   1:  PR[91,3] = PR[90,3] + 50.738;
   1:L PR[91] R[100]mm/sec CNT100;
   1:  PR[91,1] = PR[90,1] + 22.641;
   1:  PR[91,2] = PR[90,2] + -11.815;
   1:  PR[91,3] = PR[90,3] + 50.748;
   1:L PR[91] R[100]mm/sec CNT100;
   1:  PR[91,1] = PR[90,1] + 23.256;
   1:  PR[91,2] = PR[90,2] + -10.902;
   1:  PR[91,3] = PR[90,3] + 50.757;
   1:L PR[91] R[100]mm/sec CNT100;
   1:  PR[91,1] = PR[90,1] + 23.822;
   1:  PR[91,2] = PR[90,2] + -9.962;
   1:  PR[91,3] = PR[90,3] + 50.767;
   1:L PR[91] R[100]mm/sec CNT100;
   1:  PR[91,1] = PR[90,1] + 24.339;
   1:  PR[91,2] = PR[90,2] + -8.997;
   1:  PR[91,3] = PR[90,3] + 50.776;
   1:L PR[91] R[100]mm/sec CNT100;
   1:  PR[91,1] = PR[90,1] + 24.805;
   1:  PR[91,2] = PR[90,2] + -8.010;
   1:  PR[91,3] = PR[90,3] + 50.785;
   1:L PR[91] R[100]mm/sec CNT100;
   1:  PR[91,1] = PR[90,1] + 25.218;
   1:  PR[91,2] = PR[90,2] + -7.005;
   1:  PR[91,3] = PR[90,3] + 50.795;
   1:L PR[91] R[100]mm/sec CNT100;
   1:  PR[91,1] = PR[90,1] + 25.578;
   1:  PR[91,2] = PR[90,2] + -5.984;
   1:  PR[91,3] = PR[90,3] + 50.804;
   1:L PR[91] R[100]mm/sec CNT100;
   1:  PR[91,1] = PR[90,1] + 25.884;
   1:  PR[91,2] = PR[90,2] + -4.948;
   1:  PR[91,3] = PR[90,3] + 50.813;
   1:L PR[91] R[100]mm/sec CNT100;
   1:  PR[91,1] = PR[90,1] + 26.135;
   1:  PR[91,2] = PR[90,2] + -3.900;
   1:  PR[91,3] = PR[90,3] + 50.822;
   1:L PR[91] R[100]mm/sec CNT100;
   1:  PR[91,1] = PR[90,1] + 26.331;
   1:  PR[91,2] = PR[90,2] + -2.838;
   1:  PR[91,3] = PR[90,3] + 50.832;
   1:L PR[91] R[100]mm/sec CNT100;
   1:  PR[91,1] = PR[90,1] + 26.472;
   1:  PR[91,2] = PR[90,2] + -1.762;
   1:  PR[91,3] = PR[90,3] + 50.841;
   1:L PR[91] R[100]mm/sec CNT100;
   1:  PR[91,1] = PR[90,1] + 26.556;
   1:  PR[91,2] = PR[90,2] + -0.674;
   1:  PR[91,3] = PR[90,3] + 50.850;
   1:L PR[91] R[100]mm/sec CNT100;
   1:  PR[91,1] = PR[90,1] + 26.584;
   1:  PR[91,2] = PR[90,2] + 0.428;
   1:  PR[91,3] = PR[90,3] + 50.860;
   1:L PR[91] R[100]mm/sec CNT100;
   1:  PR[91,1] = PR[90,1] + 26.556;
   1:  PR[91,2] = PR[90,2] + 1.529;
   1:  PR[91,3] = PR[90,3] + 50.869;
   1:L PR[91] R[100]mm/sec CNT100;
   1:  PR[91,1] = PR[90,1] + 26.472;
   1:  PR[91,2] = PR[90,2] + 2.617;
   1:  PR[91,3] = PR[90,3] + 50.878;
   1:L PR[91] R[100]mm/sec CNT100;
   1:  PR[91,1] = PR[90,1] + 26.331;
   1:  PR[91,2] = PR[90,2] + 3.692;
   1:  PR[91,3] = PR[90,3] + 50.888;
   1:L PR[91] R[100]mm/sec CNT100;
   1:  PR[91,1] = PR[90,1] + 26.135;
   1:  PR[91,2] = PR[90,2] + 4.755;
   1:  PR[91,3] = PR[90,3] + 50.897;
   1:L PR[91] R[100]mm/sec CNT100;
   1:  PR[91,1] = PR[90,1] + 25.884;
   1:  PR[91,2] = PR[90,2] + 5.803;
   1:  PR[91,3] = PR[90,3] + 50.906;
   1:L PR[91] R[100]mm/sec CNT100;
   1:  PR[91,1] = PR[90,1] + 25.578;
   1:  PR[91,2] = PR[90,2] + 6.839;
   1:  PR[91,3] = PR[90,3] + 50.915;
   1:L PR[91] R[100]mm/sec CNT100;
   1:  PR[91,1] = PR[90,1] + 25.218;
   1:  PR[91,2] = PR[90,2] + 7.860;
   1:  PR[91,3] = PR[90,3] + 50.925;
   1:L PR[91] R[100]mm/sec CNT100;
   1:  PR[91,1] = PR[90,1] + 24.805;
   1:  PR[91,2] = PR[90,2] + 8.864;
   1:  PR[91,3] = PR[90,3] + 50.934;
   1:L PR[91] R[100]mm/sec CNT100;
   1:  PR[91,1] = PR[90,1] + 24.339;
   1:  PR[91,2] = PR[90,2] + 9.851;
   1:  PR[91,3] = PR[90,3] + 50.943;
   1:L PR[91] R[100]mm/sec CNT100;
   1:  PR[91,1] = PR[90,1] + 23.823;
   1:  PR[91,2] = PR[90,2] + 10.817;
   1:  PR[91,3] = PR[90,3] + 50.953;
   1:L PR[91] R[100]mm/sec CNT100;
   1:  PR[91,1] = PR[90,1] + 23.256;
   1:  PR[91,2] = PR[90,2] + 11.757;
   1:  PR[91,3] = PR[90,3] + 50.962;
   1:L PR[91] R[100]mm/sec CNT100;
   1:  PR[91,1] = PR[90,1] + 22.642;
   1:  PR[91,2] = PR[90,2] + 12.669;
   1:  PR[91,3] = PR[90,3] + 50.971;
   1:L PR[91] R[100]mm/sec CNT100;
   1:  PR[91,1] = PR[90,1] + 21.980;
   1:  PR[91,2] = PR[90,2] + 13.551;
   1:  PR[91,3] = PR[90,3] + 50.981;
   1:L PR[91] R[100]mm/sec CNT100;
   1:  PR[91,1] = PR[90,1] + 21.273;
   1:  PR[91,2] = PR[90,2] + 14.398;
   1:  PR[91,3] = PR[90,3] + 50.990;
   1:L PR[91] R[100]mm/sec CNT100;
   1:  PR[91,1] = PR[90,1] + 20.523;
   1:  PR[91,2] = PR[90,2] + 15.210;
   1:  PR[91,3] = PR[90,3] + 51.000;
   1:L PR[91] R[100]mm/sec CNT100;
   1:  PR[91,1] = PR[90,1] + 19.731;
   1:  PR[91,2] = PR[90,2] + 15.984;
   1:  PR[91,3] = PR[90,3] + 51.009;
   1:L PR[91] R[100]mm/sec CNT100;
   1:  PR[91,1] = PR[90,1] + 18.899;
   1:  PR[91,2] = PR[90,2] + 16.718;
   1:  PR[91,3] = PR[90,3] + 51.019;
   1:L PR[91] R[100]mm/sec CNT100;
   1:  PR[91,1] = PR[90,1] + 18.029;
   1:  PR[91,2] = PR[90,2] + 17.410;
   1:  PR[91,3] = PR[90,3] + 51.028;
   1:L PR[91] R[100]mm/sec CNT100;
   1:  PR[91,1] = PR[90,1] + 17.123;
   1:  PR[91,2] = PR[90,2] + 18.058;
   1:  PR[91,3] = PR[90,3] + 51.038;
   1:L PR[91] R[100]mm/sec CNT100;
   1:  PR[91,1] = PR[90,1] + 16.184;
   1:  PR[91,2] = PR[90,2] + 18.663;
   1:  PR[91,3] = PR[90,3] + 51.047;
   1:L PR[91] R[100]mm/sec CNT100;
   1:  PR[91,1] = PR[90,1] + 15.213;
   1:  PR[91,2] = PR[90,2] + 19.221;
   1:  PR[91,3] = PR[90,3] + 51.057;
   1:L PR[91] R[100]mm/sec CNT100;
   1:  PR[91,1] = PR[90,1] + 14.214;
   1:  PR[91,2] = PR[90,2] + 19.731;
   1:  PR[91,3] = PR[90,3] + 51.066;
   1:L PR[91] R[100]mm/sec CNT100;
   1:  PR[91,1] = PR[90,1] + 13.188;
   1:  PR[91,2] = PR[90,2] + 20.191;
   1:  PR[91,3] = PR[90,3] + 51.076;
   1:L PR[91] R[100]mm/sec CNT100;
   1:  PR[91,1] = PR[90,1] + 12.139;
   1:  PR[91,2] = PR[90,2] + 20.599;
   1:  PR[91,3] = PR[90,3] + 51.085;
   1:L PR[91] R[100]mm/sec CNT100;
   1:  PR[91,1] = PR[90,1] + 11.070;
   1:  PR[91,2] = PR[90,2] + 20.955;
   1:  PR[91,3] = PR[90,3] + 51.095;
   1:L PR[91] R[100]mm/sec CNT100;
   1:  PR[91,1] = PR[90,1] + 9.982;
   1:  PR[91,2] = PR[90,2] + 21.257;
   1:  PR[91,3] = PR[90,3] + 51.105;
   1:L PR[91] R[100]mm/sec CNT100;
   1:  PR[91,1] = PR[90,1] + 8.879;
   1:  PR[91,2] = PR[90,2] + 21.504;
   1:  PR[91,3] = PR[90,3] + 51.114;
   1:L PR[91] R[100]mm/sec CNT100;
   1:  PR[91,1] = PR[90,1] + 7.764;
   1:  PR[91,2] = PR[90,2] + 21.696;
   1:  PR[91,3] = PR[90,3] + 51.124;
   1:L PR[91] R[100]mm/sec CNT100;
   1:  PR[91,1] = PR[90,1] + 6.640;
   1:  PR[91,2] = PR[90,2] + 21.831;
   1:  PR[91,3] = PR[90,3] + 51.134;
   1:L PR[91] R[100]mm/sec CNT100;
   1:  PR[91,1] = PR[90,1] + 5.508;
   1:  PR[91,2] = PR[90,2] + 21.910;
   1:  PR[91,3] = PR[90,3] + 51.143;
   1:L PR[91] R[100]mm/sec CNT100;
   1:  PR[91,1] = PR[90,1] + 4.806;
   1:  PR[91,2] = PR[90,2] + 21.924;
   1:  PR[91,3] = PR[90,3] + 51.153;
   1:L PR[91] R[100]mm/sec CNT100;
   1:  PR[91,1] = PR[90,1] + 4.375;
   1:  PR[91,2] = PR[90,2] + 21.931;
   1:  PR[91,3] = PR[90,3] + 51.159;
   1:L PR[91] R[100]mm/sec CNT100;
   1:  PR[91,1] = PR[90,1] + 3.240;
   1:  PR[91,2] = PR[90,2] + 21.895;
   1:  PR[91,3] = PR[90,3] + 51.163;
   1:L PR[91] R[100]mm/sec CNT100;
   1:  PR[91,1] = PR[90,1] + 2.109;
   1:  PR[91,2] = PR[90,2] + 21.801;
   1:  PR[91,3] = PR[90,3] + 51.173;
   1:L PR[91] R[100]mm/sec CNT100;
   1:  PR[91,1] = PR[90,1] + 0.962;
   1:  PR[91,2] = PR[90,2] + 21.646;
   1:  PR[91,3] = PR[90,3] + 51.182;
   1:L PR[91] R[100]mm/sec CNT100;
   1:  PR[91,1] = PR[90,1] + 0.291;
   1:  PR[91,2] = PR[90,2] + 21.527;
   1:  PR[91,3] = PR[90,3] + 51.192;
   1:L PR[91] R[100]mm/sec CNT100;
   1:  PR[91,1] = PR[90,1] + -0.185;
   1:  PR[91,2] = PR[90,2] + 21.498;
   1:  PR[91,3] = PR[90,3] + 51.198;
   1:L PR[91] R[100]mm/sec CNT100;
   1:  PR[91,1] = PR[90,1] + -0.645;
   1:  PR[91,2] = PR[90,2] + 21.546;
   1:  PR[91,3] = PR[90,3] + 51.202;
   1:L PR[91] R[100]mm/sec CNT100;
   1:  PR[91,1] = PR[90,1] + -1.218;
   1:  PR[91,2] = PR[90,2] + 21.650;
   1:  PR[91,3] = PR[90,3] + 51.206;
   1:L PR[91] R[100]mm/sec CNT100;
   1:  PR[91,1] = PR[90,1] + -2.346;
   1:  PR[91,2] = PR[90,2] + 21.801;
   1:  PR[91,3] = PR[90,3] + 51.211;
   1:L PR[91] R[100]mm/sec CNT100;
   1:  PR[91,1] = PR[90,1] + -3.478;
   1:  PR[91,2] = PR[90,2] + 21.895;
   1:  PR[91,3] = PR[90,3] + 51.221;
   1:L PR[91] R[100]mm/sec CNT100;
   1:  PR[91,1] = PR[90,1] + -4.612;
   1:  PR[91,2] = PR[90,2] + 21.931;
   1:  PR[91,3] = PR[90,3] + 51.230;
   1:L PR[91] R[100]mm/sec CNT100;
   1:  PR[91,1] = PR[90,1] + -5.746;
   1:  PR[91,2] = PR[90,2] + 21.909;
   1:  PR[91,3] = PR[90,3] + 51.240;
   1:L PR[91] R[100]mm/sec CNT100;
   1:  PR[91,1] = PR[90,1] + -6.877;
   1:  PR[91,2] = PR[90,2] + 21.831;
   1:  PR[91,3] = PR[90,3] + 51.250;
   1:L PR[91] R[100]mm/sec CNT100;
   1:  PR[91,1] = PR[90,1] + -8.001;
   1:  PR[91,2] = PR[90,2] + 21.696;
   1:  PR[91,3] = PR[90,3] + 51.260;
   1:L PR[91] R[100]mm/sec CNT100;
   1:  PR[91,1] = PR[90,1] + -9.117;
   1:  PR[91,2] = PR[90,2] + 21.504;
   1:  PR[91,3] = PR[90,3] + 51.269;
   1:L PR[91] R[100]mm/sec CNT100;
   1:  PR[91,1] = PR[90,1] + -10.219;
   1:  PR[91,2] = PR[90,2] + 21.257;
   1:  PR[91,3] = PR[90,3] + 51.279;
   1:L PR[91] R[100]mm/sec CNT100;
   1:  PR[91,1] = PR[90,1] + -11.307;
   1:  PR[91,2] = PR[90,2] + 20.955;
   1:  PR[91,3] = PR[90,3] + 51.289;
   1:L PR[91] R[100]mm/sec CNT100;
   1:  PR[91,1] = PR[90,1] + -12.377;
   1:  PR[91,2] = PR[90,2] + 20.600;
   1:  PR[91,3] = PR[90,3] + 51.298;
   1:L PR[91] R[100]mm/sec CNT100;
   1:  PR[91,1] = PR[90,1] + -13.426;
   1:  PR[91,2] = PR[90,2] + 20.191;
   1:  PR[91,3] = PR[90,3] + 51.308;
   1:L PR[91] R[100]mm/sec CNT100;
   1:  PR[91,1] = PR[90,1] + -14.451;
   1:  PR[91,2] = PR[90,2] + 19.731;
   1:  PR[91,3] = PR[90,3] + 51.318;
   1:L PR[91] R[100]mm/sec CNT100;
   1:  PR[91,1] = PR[90,1] + -15.450;
   1:  PR[91,2] = PR[90,2] + 19.222;
   1:  PR[91,3] = PR[90,3] + 51.327;
   1:L PR[91] R[100]mm/sec CNT100;
   1:  PR[91,1] = PR[90,1] + -16.421;
   1:  PR[91,2] = PR[90,2] + 18.663;
   1:  PR[91,3] = PR[90,3] + 51.337;
   1:L PR[91] R[100]mm/sec CNT100;
   1:  PR[91,1] = PR[90,1] + -17.362;
   1:  PR[91,2] = PR[90,2] + 18.057;
   1:  PR[91,3] = PR[90,3] + 51.346;
   1:L PR[91] R[100]mm/sec CNT100;
   1:  PR[91,1] = PR[90,1] + -18.267;
   1:  PR[91,2] = PR[90,2] + 17.409;
   1:  PR[91,3] = PR[90,3] + 51.356;
   1:L PR[91] R[100]mm/sec CNT100;
   1:  PR[91,1] = PR[90,1] + -19.137;
   1:  PR[91,2] = PR[90,2] + 16.717;
   1:  PR[91,3] = PR[90,3] + 51.365;
   1:L PR[91] R[100]mm/sec CNT100;
   1:  PR[91,1] = PR[90,1] + -19.969;
   1:  PR[91,2] = PR[90,2] + 15.984;
   1:  PR[91,3] = PR[90,3] + 51.375;
   1:L PR[91] R[100]mm/sec CNT100;
   1:  PR[91,1] = PR[90,1] + -20.761;
   1:  PR[91,2] = PR[90,2] + 15.211;
   1:  PR[91,3] = PR[90,3] + 51.384;
   1:L PR[91] R[100]mm/sec CNT100;
   1:  PR[91,1] = PR[90,1] + -21.512;
   1:  PR[91,2] = PR[90,2] + 14.400;
   1:  PR[91,3] = PR[90,3] + 51.394;
   1:L PR[91] R[100]mm/sec CNT100;
   1:  PR[91,1] = PR[90,1] + -22.219;
   1:  PR[91,2] = PR[90,2] + 13.553;
   1:  PR[91,3] = PR[90,3] + 51.403;
   1:L PR[91] R[100]mm/sec CNT100;
   1:  PR[91,1] = PR[90,1] + -22.880;
   1:  PR[91,2] = PR[90,2] + 12.672;
   1:  PR[91,3] = PR[90,3] + 51.413;
   1:L PR[91] R[100]mm/sec CNT100;
   1:  PR[91,1] = PR[90,1] + -23.495;
   1:  PR[91,2] = PR[90,2] + 11.760;
   1:  PR[91,3] = PR[90,3] + 51.422;
   1:L PR[91] R[100]mm/sec CNT100;
   1:  PR[91,1] = PR[90,1] + -24.061;
   1:  PR[91,2] = PR[90,2] + 10.819;
   1:  PR[91,3] = PR[90,3] + 51.432;
   1:L PR[91] R[100]mm/sec CNT100;
   1:  PR[91,1] = PR[90,1] + -24.577;
   1:  PR[91,2] = PR[90,2] + 9.853;
   1:  PR[91,3] = PR[90,3] + 51.441;
   1:L PR[91] R[100]mm/sec CNT100;
   1:  PR[91,1] = PR[90,1] + -25.043;
   1:  PR[91,2] = PR[90,2] + 8.864;
   1:  PR[91,3] = PR[90,3] + 51.450;
   1:L PR[91] R[100]mm/sec CNT100;
   1:  PR[91,1] = PR[90,1] + -25.456;
   1:  PR[91,2] = PR[90,2] + 7.857;
   1:  PR[91,3] = PR[90,3] + 51.460;
   1:L PR[91] R[100]mm/sec CNT100;
   1:  PR[91,1] = PR[90,1] + -25.816;
   1:  PR[91,2] = PR[90,2] + 6.834;
   1:  PR[91,3] = PR[90,3] + 51.469;
   1:L PR[91] R[100]mm/sec CNT100;
   1:  PR[91,1] = PR[90,1] + -26.122;
   1:  PR[91,2] = PR[90,2] + 5.798;
   1:  PR[91,3] = PR[90,3] + 51.478;
   1:L PR[91] R[100]mm/sec CNT100;
   1:  PR[91,1] = PR[90,1] + -26.374;
   1:  PR[91,2] = PR[90,2] + 4.750;
   1:  PR[91,3] = PR[90,3] + 51.488;
   1:L PR[91] R[100]mm/sec CNT100;
   1:  PR[91,1] = PR[90,1] + -26.570;
   1:  PR[91,2] = PR[90,2] + 3.689;
   1:  PR[91,3] = PR[90,3] + 51.497;
   1:L PR[91] R[100]mm/sec CNT100;
   1:  PR[91,1] = PR[90,1] + -26.710;
   1:  PR[91,2] = PR[90,2] + 2.615;
   1:  PR[91,3] = PR[90,3] + 51.506;
   1:L PR[91] R[100]mm/sec CNT100;
   1:  PR[91,1] = PR[90,1] + -26.795;
   1:  PR[91,2] = PR[90,2] + 1.528;
   1:  PR[91,3] = PR[90,3] + 51.515;
   1:L PR[91] R[100]mm/sec CNT100;
   1:  PR[91,1] = PR[90,1] + -26.823;
   1:  PR[91,2] = PR[90,2] + 0.428;
   1:  PR[91,3] = PR[90,3] + 51.525;
   1:L PR[91] R[100]mm/sec CNT100;
   1:  PR[91,1] = PR[90,1] + -26.795;
   1:  PR[91,2] = PR[90,2] + -0.673;
   1:  PR[91,3] = PR[90,3] + 51.534;
   1:L PR[91] R[100]mm/sec CNT100;
   1:  PR[91,1] = PR[90,1] + -26.710;
   1:  PR[91,2] = PR[90,2] + -1.760;
   1:  PR[91,3] = PR[90,3] + 51.543;
   1:L PR[91] R[100]mm/sec CNT100;
   1:  PR[91,1] = PR[90,1] + -26.570;
   1:  PR[91,2] = PR[90,2] + -2.834;
   1:  PR[91,3] = PR[90,3] + 51.553;
   1:L PR[91] R[100]mm/sec CNT100;
   1:  PR[91,1] = PR[90,1] + -26.374;
   1:  PR[91,2] = PR[90,2] + -3.895;
   1:  PR[91,3] = PR[90,3] + 51.562;
   1:L PR[91] R[100]mm/sec CNT100;
   1:  PR[91,1] = PR[90,1] + -26.122;
   1:  PR[91,2] = PR[90,2] + -4.944;
   1:  PR[91,3] = PR[90,3] + 51.571;
   1:L PR[91] R[100]mm/sec CNT100;
   1:  PR[91,1] = PR[90,1] + -25.816;
   1:  PR[91,2] = PR[90,2] + -5.980;
   1:  PR[91,3] = PR[90,3] + 51.580;
   1:L PR[91] R[100]mm/sec CNT100;
   1:  PR[91,1] = PR[90,1] + -25.456;
   1:  PR[91,2] = PR[90,2] + -7.002;
   1:  PR[91,3] = PR[90,3] + 51.590;
   1:L PR[91] R[100]mm/sec CNT100;
   1:  PR[91,1] = PR[90,1] + -25.043;
   1:  PR[91,2] = PR[90,2] + -8.010;
   1:  PR[91,3] = PR[90,3] + 51.599;
   1:L PR[91] R[100]mm/sec CNT100;
   1:  PR[91,1] = PR[90,1] + -24.577;
   1:  PR[91,2] = PR[90,2] + -8.998;
   1:  PR[91,3] = PR[90,3] + 51.608;
   1:L PR[91] R[100]mm/sec CNT100;
   1:  PR[91,1] = PR[90,1] + -24.061;
   1:  PR[91,2] = PR[90,2] + -9.965;
   1:  PR[91,3] = PR[90,3] + 51.618;
   1:L PR[91] R[100]mm/sec CNT100;
   1:  PR[91,1] = PR[90,1] + -23.494;
   1:  PR[91,2] = PR[90,2] + -10.906;
   1:  PR[91,3] = PR[90,3] + 51.627;
   1:L PR[91] R[100]mm/sec CNT100;
   1:  PR[91,1] = PR[90,1] + -22.880;
   1:  PR[91,2] = PR[90,2] + -11.818;
   1:  PR[91,3] = PR[90,3] + 51.636;
   1:L PR[91] R[100]mm/sec CNT100;
   1:  PR[91,1] = PR[90,1] + -22.218;
   1:  PR[91,2] = PR[90,2] + -12.698;
   1:  PR[91,3] = PR[90,3] + 51.646;
   1:L PR[91] R[100]mm/sec CNT100;
   1:  PR[91,1] = PR[90,1] + -21.511;
   1:  PR[91,2] = PR[90,2] + -13.545;
   1:  PR[91,3] = PR[90,3] + 51.655;
   1:L PR[91] R[100]mm/sec CNT100;
   1:  PR[91,1] = PR[90,1] + -20.760;
   1:  PR[91,2] = PR[90,2] + -14.356;
   1:  PR[91,3] = PR[90,3] + 51.665;
   1:L PR[91] R[100]mm/sec CNT100;
   1:  PR[91,1] = PR[90,1] + -19.968;
   1:  PR[91,2] = PR[90,2] + -15.129;
   1:  PR[91,3] = PR[90,3] + 51.674;
   1:L PR[91] R[100]mm/sec CNT100;
   1:  PR[91,1] = PR[90,1] + -19.136;
   1:  PR[91,2] = PR[90,2] + -15.863;
   1:  PR[91,3] = PR[90,3] + 51.684;
   1:L PR[91] R[100]mm/sec CNT100;
   1:  PR[91,1] = PR[90,1] + -18.266;
   1:  PR[91,2] = PR[90,2] + -16.555;
   1:  PR[91,3] = PR[90,3] + 51.693;
   1:L PR[91] R[100]mm/sec CNT100;
   1:  PR[91,1] = PR[90,1] + -17.360;
   1:  PR[91,2] = PR[90,2] + -17.204;
   1:  PR[91,3] = PR[90,3] + 51.703;
   1:L PR[91] R[100]mm/sec CNT100;
   1:  PR[91,1] = PR[90,1] + -16.420;
   1:  PR[91,2] = PR[90,2] + -17.809;
   1:  PR[91,3] = PR[90,3] + 51.712;
   1:L PR[91] R[100]mm/sec CNT100;
   1:  PR[91,1] = PR[90,1] + -15.449;
   1:  PR[91,2] = PR[90,2] + -18.367;
   1:  PR[91,3] = PR[90,3] + 51.722;
   1:L PR[91] R[100]mm/sec CNT100;
   1:  PR[91,1] = PR[90,1] + -14.450;
   1:  PR[91,2] = PR[90,2] + -18.877;
   1:  PR[91,3] = PR[90,3] + 51.731;
   1:L PR[91] R[100]mm/sec CNT100;
   1:  PR[91,1] = PR[90,1] + -13.424;
   1:  PR[91,2] = PR[90,2] + -19.337;
   1:  PR[91,3] = PR[90,3] + 51.741;
   1:L PR[91] R[100]mm/sec CNT100;
   1:  PR[91,1] = PR[90,1] + -12.375;
   1:  PR[91,2] = PR[90,2] + -19.745;
   1:  PR[91,3] = PR[90,3] + 51.750;
   1:L PR[91] R[100]mm/sec CNT100;
   1:  PR[91,1] = PR[90,1] + -11.305;
   1:  PR[91,2] = PR[90,2] + -20.101;
   1:  PR[91,3] = PR[90,3] + 51.760;
   1:L PR[91] R[100]mm/sec CNT100;
   1:  PR[91,1] = PR[90,1] + -10.217;
   1:  PR[91,2] = PR[90,2] + -20.403;
   1:  PR[91,3] = PR[90,3] + 51.770;
   1:L PR[91] R[100]mm/sec CNT100;
   1:  PR[91,1] = PR[90,1] + -9.114;
   1:  PR[91,2] = PR[90,2] + -20.650;
   1:  PR[91,3] = PR[90,3] + 51.779;
   1:L PR[91] R[100]mm/sec CNT100;
   1:  PR[91,1] = PR[90,1] + -7.999;
   1:  PR[91,2] = PR[90,2] + -20.841;
   1:  PR[91,3] = PR[90,3] + 51.789;
   1:L PR[91] R[100]mm/sec CNT100;
   1:  PR[91,1] = PR[90,1] + -6.874;
   1:  PR[91,2] = PR[90,2] + -20.976;
   1:  PR[91,3] = PR[90,3] + 51.799;
   1:L PR[91] R[100]mm/sec CNT100;
   1:  PR[91,1] = PR[90,1] + -5.742;
   1:  PR[91,2] = PR[90,2] + -21.055;
   1:  PR[91,3] = PR[90,3] + 51.808;
   1:L PR[91] R[100]mm/sec CNT100;
   1:  PR[91,1] = PR[90,1] + -5.040;
   1:  PR[91,2] = PR[90,2] + -21.069;
   1:  PR[91,3] = PR[90,3] + 51.818;
   1:L PR[91] R[100]mm/sec CNT100;
   1:  PR[91,1] = PR[90,1] + -4.609;
   1:  PR[91,2] = PR[90,2] + -21.076;
   1:  PR[91,3] = PR[90,3] + 51.824;
   1:L PR[91] R[100]mm/sec CNT100;
   1:  PR[91,1] = PR[90,1] + -3.474;
   1:  PR[91,2] = PR[90,2] + -21.039;
   1:  PR[91,3] = PR[90,3] + 51.828;
   1:L PR[91] R[100]mm/sec CNT100;
   1:  PR[91,1] = PR[90,1] + -2.342;
   1:  PR[91,2] = PR[90,2] + -20.945;
   1:  PR[91,3] = PR[90,3] + 51.838;
   1:L PR[91] R[100]mm/sec CNT100;
   1:  PR[91,1] = PR[90,1] + -1.212;
   1:  PR[91,2] = PR[90,2] + -20.793;
   1:  PR[91,3] = PR[90,3] + 51.847;
   1:L PR[91] R[100]mm/sec CNT100;
   1:  PR[91,1] = PR[90,1] + -0.645;
   1:  PR[91,2] = PR[90,2] + -20.691;
   1:  PR[91,3] = PR[90,3] + 51.857;
   1:L PR[91] R[100]mm/sec CNT100;
   1:  PR[91,1] = PR[90,1] + -0.185;
   1:  PR[91,2] = PR[90,2] + -20.643;
   1:  PR[91,3] = PR[90,3] + 51.862;
   1:L PR[91] R[100]mm/sec CNT100;
   1:  PR[91,1] = PR[90,1] + 0.291;
   1:  PR[91,2] = PR[90,2] + -20.672;
   1:  PR[91,3] = PR[90,3] + 51.866;
   1:L PR[91] R[100]mm/sec CNT100;
   1:  PR[91] = PR[90];
   1:  PR[91,1] = PR[90,1] + 1.550;
   1:  PR[91,2] = PR[90,2] + -21.205;
   1:  PR[91,3] = PR[90,3] + 53.200;
   1:L PR[91] R[100]mm/sec CNT100;
   1:  PR[91,1] = PR[90,1] + 2.692;
   1:  PR[91,2] = PR[90,2] + -21.302;
   1:  PR[91,3] = PR[90,3] + 51.880;
   1:L PR[91] R[100]mm/sec CNT100;
   1:  PR[91,1] = PR[90,1] + 3.838;
   1:  PR[91,2] = PR[90,2] + -21.341;
   1:  PR[91,3] = PR[90,3] + 51.890;
   1:L PR[91] R[100]mm/sec CNT100;
   1:  PR[91,1] = PR[90,1] + 4.984;
   1:  PR[91,2] = PR[90,2] + -21.322;
   1:  PR[91,3] = PR[90,3] + 51.900;
   1:L PR[91] R[100]mm/sec CNT100;
   1:  PR[91,1] = PR[90,1] + 6.126;
   1:  PR[91,2] = PR[90,2] + -21.245;
   1:  PR[91,3] = PR[90,3] + 51.910;
   1:L PR[91] R[100]mm/sec CNT100;
   1:  PR[91,1] = PR[90,1] + 7.262;
   1:  PR[91,2] = PR[90,2] + -21.111;
   1:  PR[91,3] = PR[90,3] + 51.920;
   1:L PR[91] R[100]mm/sec CNT100;
   1:  PR[91,1] = PR[90,1] + 8.389;
   1:  PR[91,2] = PR[90,2] + -20.919;
   1:  PR[91,3] = PR[90,3] + 51.930;
   1:L PR[91] R[100]mm/sec CNT100;
   1:  PR[91,1] = PR[90,1] + 9.504;
   1:  PR[91,2] = PR[90,2] + -20.671;
   1:  PR[91,3] = PR[90,3] + 51.939;
   1:L PR[91] R[100]mm/sec CNT100;
   1:  PR[91,1] = PR[90,1] + 10.604;
   1:  PR[91,2] = PR[90,2] + -20.367;
   1:  PR[91,3] = PR[90,3] + 51.949;
   1:L PR[91] R[100]mm/sec CNT100;
   1:  PR[91,1] = PR[90,1] + 11.685;
   1:  PR[91,2] = PR[90,2] + -20.009;
   1:  PR[91,3] = PR[90,3] + 51.959;
   1:L PR[91] R[100]mm/sec CNT100;
   1:  PR[91,1] = PR[90,1] + 12.746;
   1:  PR[91,2] = PR[90,2] + -19.597;
   1:  PR[91,3] = PR[90,3] + 51.969;
   1:L PR[91] R[100]mm/sec CNT100;
   1:  PR[91,1] = PR[90,1] + 13.783;
   1:  PR[91,2] = PR[90,2] + -19.134;
   1:  PR[91,3] = PR[90,3] + 51.979;
   1:L PR[91] R[100]mm/sec CNT100;
   1:  PR[91,1] = PR[90,1] + 14.794;
   1:  PR[91,2] = PR[90,2] + -18.619;
   1:  PR[91,3] = PR[90,3] + 51.988;
   1:L PR[91] R[100]mm/sec CNT100;
   1:  PR[91,1] = PR[90,1] + 15.776;
   1:  PR[91,2] = PR[90,2] + -18.055;
   1:  PR[91,3] = PR[90,3] + 51.998;
   1:L PR[91] R[100]mm/sec CNT100;
   1:  PR[91,1] = PR[90,1] + 16.727;
   1:  PR[91,2] = PR[90,2] + -17.444;
   1:  PR[91,3] = PR[90,3] + 52.008;
   1:L PR[91] R[100]mm/sec CNT100;
   1:  PR[91,1] = PR[90,1] + 17.643;
   1:  PR[91,2] = PR[90,2] + -16.787;
   1:  PR[91,3] = PR[90,3] + 52.017;
   1:L PR[91] R[100]mm/sec CNT100;
   1:  PR[91,1] = PR[90,1] + 18.524;
   1:  PR[91,2] = PR[90,2] + -16.086;
   1:  PR[91,3] = PR[90,3] + 52.027;
   1:L PR[91] R[100]mm/sec CNT100;
   1:  PR[91,1] = PR[90,1] + 19.366;
   1:  PR[91,2] = PR[90,2] + -15.342;
   1:  PR[91,3] = PR[90,3] + 52.037;
   1:L PR[91] R[100]mm/sec CNT100;
   1:  PR[91,1] = PR[90,1] + 20.168;
   1:  PR[91,2] = PR[90,2] + -14.558;
   1:  PR[91,3] = PR[90,3] + 52.046;
   1:L PR[91] R[100]mm/sec CNT100;
   1:  PR[91,1] = PR[90,1] + 20.928;
   1:  PR[91,2] = PR[90,2] + -13.735;
   1:  PR[91,3] = PR[90,3] + 52.056;
   1:L PR[91] R[100]mm/sec CNT100;
   1:  PR[91,1] = PR[90,1] + 21.643;
   1:  PR[91,2] = PR[90,2] + -12.876;
   1:  PR[91,3] = PR[90,3] + 52.066;
   1:L PR[91] R[100]mm/sec CNT100;
   1:  PR[91,1] = PR[90,1] + 22.312;
   1:  PR[91,2] = PR[90,2] + -11.983;
   1:  PR[91,3] = PR[90,3] + 52.075;
   1:L PR[91] R[100]mm/sec CNT100;
   1:  PR[91,1] = PR[90,1] + 22.934;
   1:  PR[91,2] = PR[90,2] + -11.058;
   1:  PR[91,3] = PR[90,3] + 52.085;
   1:L PR[91] R[100]mm/sec CNT100;
   1:  PR[91,1] = PR[90,1] + 23.507;
   1:  PR[91,2] = PR[90,2] + -10.105;
   1:  PR[91,3] = PR[90,3] + 52.094;
   1:L PR[91] R[100]mm/sec CNT100;
   1:  PR[91,1] = PR[90,1] + 24.030;
   1:  PR[91,2] = PR[90,2] + -9.127;
   1:  PR[91,3] = PR[90,3] + 52.104;
   1:L PR[91] R[100]mm/sec CNT100;
   1:  PR[91,1] = PR[90,1] + 24.501;
   1:  PR[91,2] = PR[90,2] + -8.126;
   1:  PR[91,3] = PR[90,3] + 52.113;
   1:L PR[91] R[100]mm/sec CNT100;
   1:  PR[91,1] = PR[90,1] + 24.919;
   1:  PR[91,2] = PR[90,2] + -7.107;
   1:  PR[91,3] = PR[90,3] + 52.123;
   1:L PR[91] R[100]mm/sec CNT100;
   1:  PR[91,1] = PR[90,1] + 25.283;
   1:  PR[91,2] = PR[90,2] + -6.071;
   1:  PR[91,3] = PR[90,3] + 52.132;
   1:L PR[91] R[100]mm/sec CNT100;
   1:  PR[91,1] = PR[90,1] + 25.592;
   1:  PR[91,2] = PR[90,2] + -5.020;
   1:  PR[91,3] = PR[90,3] + 52.142;
   1:L PR[91] R[100]mm/sec CNT100;
   1:  PR[91,1] = PR[90,1] + 25.846;
   1:  PR[91,2] = PR[90,2] + -3.955;
   1:  PR[91,3] = PR[90,3] + 52.151;
   1:L PR[91] R[100]mm/sec CNT100;
   1:  PR[91,1] = PR[90,1] + 26.045;
   1:  PR[91,2] = PR[90,2] + -2.877;
   1:  PR[91,3] = PR[90,3] + 52.161;
   1:L PR[91] R[100]mm/sec CNT100;
   1:  PR[91,1] = PR[90,1] + 26.187;
   1:  PR[91,2] = PR[90,2] + -1.787;
   1:  PR[91,3] = PR[90,3] + 52.170;
   1:L PR[91] R[100]mm/sec CNT100;
   1:  PR[91,1] = PR[90,1] + 26.272;
   1:  PR[91,2] = PR[90,2] + -0.686;
   1:  PR[91,3] = PR[90,3] + 52.179;
   1:L PR[91] R[100]mm/sec CNT100;
   1:  PR[91,1] = PR[90,1] + 26.298;
   1:  PR[91,2] = PR[90,2] + 0.428;
   1:  PR[91,3] = PR[90,3] + 52.189;
   1:L PR[91] R[100]mm/sec CNT100;
   1:  PR[91,1] = PR[90,1] + 26.272;
   1:  PR[91,2] = PR[90,2] + 1.541;
   1:  PR[91,3] = PR[90,3] + 52.198;
   1:L PR[91] R[100]mm/sec CNT100;
   1:  PR[91,1] = PR[90,1] + 26.187;
   1:  PR[91,2] = PR[90,2] + 2.642;
   1:  PR[91,3] = PR[90,3] + 52.208;
   1:L PR[91] R[100]mm/sec CNT100;
   1:  PR[91,1] = PR[90,1] + 26.045;
   1:  PR[91,2] = PR[90,2] + 3.732;
   1:  PR[91,3] = PR[90,3] + 52.218;
   1:L PR[91] R[100]mm/sec CNT100;
   1:  PR[91,1] = PR[90,1] + 25.846;
   1:  PR[91,2] = PR[90,2] + 4.810;
   1:  PR[91,3] = PR[90,3] + 52.227;
   1:L PR[91] R[100]mm/sec CNT100;
   1:  PR[91,1] = PR[90,1] + 25.592;
   1:  PR[91,2] = PR[90,2] + 5.874;
   1:  PR[91,3] = PR[90,3] + 52.236;
   1:L PR[91] R[100]mm/sec CNT100;
   1:  PR[91,1] = PR[90,1] + 25.283;
   1:  PR[91,2] = PR[90,2] + 6.925;
   1:  PR[91,3] = PR[90,3] + 52.246;
   1:L PR[91] R[100]mm/sec CNT100;
   1:  PR[91,1] = PR[90,1] + 24.919;
   1:  PR[91,2] = PR[90,2] + 7.961;
   1:  PR[91,3] = PR[90,3] + 52.255;
   1:L PR[91] R[100]mm/sec CNT100;
   1:  PR[91,1] = PR[90,1] + 24.501;
   1:  PR[91,2] = PR[90,2] + 8.980;
   1:  PR[91,3] = PR[90,3] + 52.265;
   1:L PR[91] R[100]mm/sec CNT100;
   1:  PR[91,1] = PR[90,1] + 24.030;
   1:  PR[91,2] = PR[90,2] + 9.981;
   1:  PR[91,3] = PR[90,3] + 52.274;
   1:L PR[91] R[100]mm/sec CNT100;
   1:  PR[91,1] = PR[90,1] + 23.508;
   1:  PR[91,2] = PR[90,2] + 10.960;
   1:  PR[91,3] = PR[90,3] + 52.284;
   1:L PR[91] R[100]mm/sec CNT100;
   1:  PR[91,1] = PR[90,1] + 22.935;
   1:  PR[91,2] = PR[90,2] + 11.912;
   1:  PR[91,3] = PR[90,3] + 52.293;
   1:L PR[91] R[100]mm/sec CNT100;
   1:  PR[91,1] = PR[90,1] + 22.313;
   1:  PR[91,2] = PR[90,2] + 12.837;
   1:  PR[91,3] = PR[90,3] + 52.303;
   1:L PR[91] R[100]mm/sec CNT100;
   1:  PR[91,1] = PR[90,1] + 21.644;
   1:  PR[91,2] = PR[90,2] + 13.730;
   1:  PR[91,3] = PR[90,3] + 52.312;
   1:L PR[91] R[100]mm/sec CNT100;
   1:  PR[91,1] = PR[90,1] + 20.929;
   1:  PR[91,2] = PR[90,2] + 14.589;
   1:  PR[91,3] = PR[90,3] + 52.322;
   1:L PR[91] R[100]mm/sec CNT100;
   1:  PR[91,1] = PR[90,1] + 20.169;
   1:  PR[91,2] = PR[90,2] + 15.412;
   1:  PR[91,3] = PR[90,3] + 52.331;
   1:L PR[91] R[100]mm/sec CNT100;
   1:  PR[91,1] = PR[90,1] + 19.367;
   1:  PR[91,2] = PR[90,2] + 16.196;
   1:  PR[91,3] = PR[90,3] + 52.341;
   1:L PR[91] R[100]mm/sec CNT100;
   1:  PR[91,1] = PR[90,1] + 18.526;
   1:  PR[91,2] = PR[90,2] + 16.939;
   1:  PR[91,3] = PR[90,3] + 52.351;
   1:L PR[91] R[100]mm/sec CNT100;
   1:  PR[91,1] = PR[90,1] + 17.645;
   1:  PR[91,2] = PR[90,2] + 17.641;
   1:  PR[91,3] = PR[90,3] + 52.360;
   1:L PR[91] R[100]mm/sec CNT100;
   1:  PR[91,1] = PR[90,1] + 16.728;
   1:  PR[91,2] = PR[90,2] + 18.298;
   1:  PR[91,3] = PR[90,3] + 52.370;
   1:L PR[91] R[100]mm/sec CNT100;
   1:  PR[91,1] = PR[90,1] + 15.778;
   1:  PR[91,2] = PR[90,2] + 18.909;
   1:  PR[91,3] = PR[90,3] + 52.380;
   1:L PR[91] R[100]mm/sec CNT100;
   1:  PR[91,1] = PR[90,1] + 14.796;
   1:  PR[91,2] = PR[90,2] + 19.473;
   1:  PR[91,3] = PR[90,3] + 52.389;
   1:L PR[91] R[100]mm/sec CNT100;
   1:  PR[91,1] = PR[90,1] + 13.786;
   1:  PR[91,2] = PR[90,2] + 19.987;
   1:  PR[91,3] = PR[90,3] + 52.399;
   1:L PR[91] R[100]mm/sec CNT100;
   1:  PR[91,1] = PR[90,1] + 12.749;
   1:  PR[91,2] = PR[90,2] + 20.451;
   1:  PR[91,3] = PR[90,3] + 52.409;
   1:L PR[91] R[100]mm/sec CNT100;
   1:  PR[91,1] = PR[90,1] + 11.688;
   1:  PR[91,2] = PR[90,2] + 20.863;
   1:  PR[91,3] = PR[90,3] + 52.418;
   1:L PR[91] R[100]mm/sec CNT100;
   1:  PR[91,1] = PR[90,1] + 10.607;
   1:  PR[91,2] = PR[90,2] + 21.221;
   1:  PR[91,3] = PR[90,3] + 52.428;
   1:L PR[91] R[100]mm/sec CNT100;
   1:  PR[91,1] = PR[90,1] + 9.508;
   1:  PR[91,2] = PR[90,2] + 21.525;
   1:  PR[91,3] = PR[90,3] + 52.438;
   1:L PR[91] R[100]mm/sec CNT100;
   1:  PR[91,1] = PR[90,1] + 8.393;
   1:  PR[91,2] = PR[90,2] + 21.773;
   1:  PR[91,3] = PR[90,3] + 52.448;
   1:L PR[91] R[100]mm/sec CNT100;
   1:  PR[91,1] = PR[90,1] + 7.266;
   1:  PR[91,2] = PR[90,2] + 21.965;
   1:  PR[91,3] = PR[90,3] + 52.458;
   1:L PR[91] R[100]mm/sec CNT100;
   1:  PR[91,1] = PR[90,1] + 6.130;
   1:  PR[91,2] = PR[90,2] + 22.100;
   1:  PR[91,3] = PR[90,3] + 52.467;
   1:L PR[91] R[100]mm/sec CNT100;
   1:  PR[91,1] = PR[90,1] + 4.988;
   1:  PR[91,2] = PR[90,2] + 22.177;
   1:  PR[91,3] = PR[90,3] + 52.477;
   1:L PR[91] R[100]mm/sec CNT100;
   1:  PR[91,1] = PR[90,1] + 3.843;
   1:  PR[91,2] = PR[90,2] + 22.197;
   1:  PR[91,3] = PR[90,3] + 52.487;
   1:L PR[91] R[100]mm/sec CNT100;
   1:  PR[91,1] = PR[90,1] + 2.697;
   1:  PR[91,2] = PR[90,2] + 22.158;
   1:  PR[91,3] = PR[90,3] + 52.497;
   1:L PR[91] R[100]mm/sec CNT100;
   1:  PR[91,1] = PR[90,1] + 1.555;
   1:  PR[91,2] = PR[90,2] + 22.061;
   1:  PR[91,3] = PR[90,3] + 52.507;
   1:L PR[91] R[100]mm/sec CNT100;
   1:  PR[91,1] = PR[90,1] + 0.328;
   1:  PR[91,2] = PR[90,2] + 21.892;
   1:  PR[91,3] = PR[90,3] + 52.517;
   1:L PR[91] R[100]mm/sec CNT100;
   1:  PR[91,1] = PR[90,1] + -0.121;
   1:  PR[91,2] = PR[90,2] + 21.856;
   1:  PR[91,3] = PR[90,3] + 52.527;
   1:L PR[91] R[100]mm/sec CNT100;
   1:  PR[91,1] = PR[90,1] + -0.576;
   1:  PR[91,2] = PR[90,2] + 21.893;
   1:  PR[91,3] = PR[90,3] + 52.531;
   1:L PR[91] R[100]mm/sec CNT100;
   1:  PR[91,1] = PR[90,1] + -1.793;
   1:  PR[91,2] = PR[90,2] + 22.061;
   1:  PR[91,3] = PR[90,3] + 52.535;
   1:L PR[91] R[100]mm/sec CNT100;
   1:  PR[91,1] = PR[90,1] + -2.935;
   1:  PR[91,2] = PR[90,2] + 22.158;
   1:  PR[91,3] = PR[90,3] + 52.545;
   1:L PR[91] R[100]mm/sec CNT100;
   1:  PR[91,1] = PR[90,1] + -4.081;
   1:  PR[91,2] = PR[90,2] + 22.196;
   1:  PR[91,3] = PR[90,3] + 52.555;
   1:L PR[91] R[100]mm/sec CNT100;
   1:  PR[91,1] = PR[90,1] + -5.226;
   1:  PR[91,2] = PR[90,2] + 22.177;
   1:  PR[91,3] = PR[90,3] + 52.565;
   1:L PR[91] R[100]mm/sec CNT100;
   1:  PR[91,1] = PR[90,1] + -6.368;
   1:  PR[91,2] = PR[90,2] + 22.100;
   1:  PR[91,3] = PR[90,3] + 52.575;
   1:L PR[91] R[100]mm/sec CNT100;
   1:  PR[91,1] = PR[90,1] + -7.504;
   1:  PR[91,2] = PR[90,2] + 21.965;
   1:  PR[91,3] = PR[90,3] + 52.585;
   1:L PR[91] R[100]mm/sec CNT100;
   1:  PR[91,1] = PR[90,1] + -8.631;
   1:  PR[91,2] = PR[90,2] + 21.773;
   1:  PR[91,3] = PR[90,3] + 52.595;
   1:L PR[91] R[100]mm/sec CNT100;
   1:  PR[91,1] = PR[90,1] + -9.746;
   1:  PR[91,2] = PR[90,2] + 21.525;
   1:  PR[91,3] = PR[90,3] + 52.604;
   1:L PR[91] R[100]mm/sec CNT100;
   1:  PR[91,1] = PR[90,1] + -10.845;
   1:  PR[91,2] = PR[90,2] + 21.222;
   1:  PR[91,3] = PR[90,3] + 52.614;
   1:L PR[91] R[100]mm/sec CNT100;
   1:  PR[91,1] = PR[90,1] + -11.926;
   1:  PR[91,2] = PR[90,2] + 20.864;
   1:  PR[91,3] = PR[90,3] + 52.624;
   1:L PR[91] R[100]mm/sec CNT100;
   1:  PR[91,1] = PR[90,1] + -12.987;
   1:  PR[91,2] = PR[90,2] + 20.452;
   1:  PR[91,3] = PR[90,3] + 52.634;
   1:L PR[91] R[100]mm/sec CNT100;
   1:  PR[91,1] = PR[90,1] + -14.024;
   1:  PR[91,2] = PR[90,2] + 19.988;
   1:  PR[91,3] = PR[90,3] + 52.644;
   1:L PR[91] R[100]mm/sec CNT100;
   1:  PR[91,1] = PR[90,1] + -15.034;
   1:  PR[91,2] = PR[90,2] + 19.473;
   1:  PR[91,3] = PR[90,3] + 52.653;
   1:L PR[91] R[100]mm/sec CNT100;
   1:  PR[91,1] = PR[90,1] + -16.016;
   1:  PR[91,2] = PR[90,2] + 18.909;
   1:  PR[91,3] = PR[90,3] + 52.663;
   1:L PR[91] R[100]mm/sec CNT100;
   1:  PR[91,1] = PR[90,1] + -16.967;
   1:  PR[91,2] = PR[90,2] + 18.298;
   1:  PR[91,3] = PR[90,3] + 52.673;
   1:L PR[91] R[100]mm/sec CNT100;
   1:  PR[91,1] = PR[90,1] + -17.883;
   1:  PR[91,2] = PR[90,2] + 17.640;
   1:  PR[91,3] = PR[90,3] + 52.682;
   1:L PR[91] R[100]mm/sec CNT100;
   1:  PR[91,1] = PR[90,1] + -18.764;
   1:  PR[91,2] = PR[90,2] + 16.939;
   1:  PR[91,3] = PR[90,3] + 52.692;
   1:L PR[91] R[100]mm/sec CNT100;
   1:  PR[91,1] = PR[90,1] + -19.606;
   1:  PR[91,2] = PR[90,2] + 16.196;
   1:  PR[91,3] = PR[90,3] + 52.702;
   1:L PR[91] R[100]mm/sec CNT100;
   1:  PR[91,1] = PR[90,1] + -20.408;
   1:  PR[91,2] = PR[90,2] + 15.412;
   1:  PR[91,3] = PR[90,3] + 52.711;
   1:L PR[91] R[100]mm/sec CNT100;
   1:  PR[91,1] = PR[90,1] + -21.167;
   1:  PR[91,2] = PR[90,2] + 14.590;
   1:  PR[91,3] = PR[90,3] + 52.721;
   1:L PR[91] R[100]mm/sec CNT100;
   1:  PR[91,1] = PR[90,1] + -21.882;
   1:  PR[91,2] = PR[90,2] + 13.732;
   1:  PR[91,3] = PR[90,3] + 52.731;
   1:L PR[91] R[100]mm/sec CNT100;
   1:  PR[91,1] = PR[90,1] + -22.551;
   1:  PR[91,2] = PR[90,2] + 12.839;
   1:  PR[91,3] = PR[90,3] + 52.740;
   1:L PR[91] R[100]mm/sec CNT100;
   1:  PR[91,1] = PR[90,1] + -23.173;
   1:  PR[91,2] = PR[90,2] + 11.915;
   1:  PR[91,3] = PR[90,3] + 52.750;
   1:L PR[91] R[100]mm/sec CNT100;
   1:  PR[91,1] = PR[90,1] + -23.746;
   1:  PR[91,2] = PR[90,2] + 10.962;
   1:  PR[91,3] = PR[90,3] + 52.759;
   1:L PR[91] R[100]mm/sec CNT100;
   1:  PR[91,1] = PR[90,1] + -24.268;
   1:  PR[91,2] = PR[90,2] + 9.983;
   1:  PR[91,3] = PR[90,3] + 52.769;
   1:L PR[91] R[100]mm/sec CNT100;
   1:  PR[91,1] = PR[90,1] + -24.739;
   1:  PR[91,2] = PR[90,2] + 8.981;
   1:  PR[91,3] = PR[90,3] + 52.778;
   1:L PR[91] R[100]mm/sec CNT100;
   1:  PR[91,1] = PR[90,1] + -25.157;
   1:  PR[91,2] = PR[90,2] + 7.959;
   1:  PR[91,3] = PR[90,3] + 52.788;
   1:L PR[91] R[100]mm/sec CNT100;
   1:  PR[91,1] = PR[90,1] + -25.521;
   1:  PR[91,2] = PR[90,2] + 6.922;
   1:  PR[91,3] = PR[90,3] + 52.797;
   1:L PR[91] R[100]mm/sec CNT100;
   1:  PR[91,1] = PR[90,1] + -25.831;
   1:  PR[91,2] = PR[90,2] + 5.870;
   1:  PR[91,3] = PR[90,3] + 52.807;
   1:L PR[91] R[100]mm/sec CNT100;
   1:  PR[91,1] = PR[90,1] + -26.085;
   1:  PR[91,2] = PR[90,2] + 4.806;
   1:  PR[91,3] = PR[90,3] + 52.816;
   1:L PR[91] R[100]mm/sec CNT100;
   1:  PR[91,1] = PR[90,1] + -26.283;
   1:  PR[91,2] = PR[90,2] + 3.729;
   1:  PR[91,3] = PR[90,3] + 52.826;
   1:L PR[91] R[100]mm/sec CNT100;
   1:  PR[91,1] = PR[90,1] + -26.425;
   1:  PR[91,2] = PR[90,2] + 2.641;
   1:  PR[91,3] = PR[90,3] + 52.835;
   1:L PR[91] R[100]mm/sec CNT100;
   1:  PR[91,1] = PR[90,1] + -26.510;
   1:  PR[91,2] = PR[90,2] + 1.541;
   1:  PR[91,3] = PR[90,3] + 52.844;
   1:L PR[91] R[100]mm/sec CNT100;
   1:  PR[91,1] = PR[90,1] + -26.537;
   1:  PR[91,2] = PR[90,2] + 0.428;
   1:  PR[91,3] = PR[90,3] + 52.854;
   1:L PR[91] R[100]mm/sec CNT100;
   1:  PR[91,1] = PR[90,1] + -26.510;
   1:  PR[91,2] = PR[90,2] + -0.686;
   1:  PR[91,3] = PR[90,3] + 52.863;
   1:L PR[91] R[100]mm/sec CNT100;
   1:  PR[91,1] = PR[90,1] + -26.425;
   1:  PR[91,2] = PR[90,2] + -1.786;
   1:  PR[91,3] = PR[90,3] + 52.873;
   1:L PR[91] R[100]mm/sec CNT100;
   1:  PR[91,1] = PR[90,1] + -26.283;
   1:  PR[91,2] = PR[90,2] + -2.874;
   1:  PR[91,3] = PR[90,3] + 52.883;
   1:L PR[91] R[100]mm/sec CNT100;
   1:  PR[91,1] = PR[90,1] + -26.085;
   1:  PR[91,2] = PR[90,2] + -3.951;
   1:  PR[91,3] = PR[90,3] + 52.892;
   1:L PR[91] R[100]mm/sec CNT100;
   1:  PR[91,1] = PR[90,1] + -25.831;
   1:  PR[91,2] = PR[90,2] + -5.015;
   1:  PR[91,3] = PR[90,3] + 52.901;
   1:L PR[91] R[100]mm/sec CNT100;
   1:  PR[91,1] = PR[90,1] + -25.521;
   1:  PR[91,2] = PR[90,2] + -6.067;
   1:  PR[91,3] = PR[90,3] + 52.911;
   1:L PR[91] R[100]mm/sec CNT100;
   1:  PR[91,1] = PR[90,1] + -25.157;
   1:  PR[91,2] = PR[90,2] + -7.105;
   1:  PR[91,3] = PR[90,3] + 52.920;
   1:L PR[91] R[100]mm/sec CNT100;
   1:  PR[91,1] = PR[90,1] + -24.739;
   1:  PR[91,2] = PR[90,2] + -8.126;
   1:  PR[91,3] = PR[90,3] + 52.930;
   1:L PR[91] R[100]mm/sec CNT100;
   1:  PR[91,1] = PR[90,1] + -24.268;
   1:  PR[91,2] = PR[90,2] + -9.128;
   1:  PR[91,3] = PR[90,3] + 52.939;
   1:L PR[91] R[100]mm/sec CNT100;
   1:  PR[91,1] = PR[90,1] + -23.745;
   1:  PR[91,2] = PR[90,2] + -10.108;
   1:  PR[91,3] = PR[90,3] + 52.949;
   1:L PR[91] R[100]mm/sec CNT100;
   1:  PR[91,1] = PR[90,1] + -23.173;
   1:  PR[91,2] = PR[90,2] + -11.061;
   1:  PR[91,3] = PR[90,3] + 52.958;
   1:L PR[91] R[100]mm/sec CNT100;
   1:  PR[91,1] = PR[90,1] + -22.551;
   1:  PR[91,2] = PR[90,2] + -11.985;
   1:  PR[91,3] = PR[90,3] + 52.968;
   1:L PR[91] R[100]mm/sec CNT100;
   1:  PR[91,1] = PR[90,1] + -21.881;
   1:  PR[91,2] = PR[90,2] + -12.878;
   1:  PR[91,3] = PR[90,3] + 52.977;
   1:L PR[91] R[100]mm/sec CNT100;
   1:  PR[91,1] = PR[90,1] + -21.166;
   1:  PR[91,2] = PR[90,2] + -13.736;
   1:  PR[91,3] = PR[90,3] + 52.987;
   1:L PR[91] R[100]mm/sec CNT100;
   1:  PR[91,1] = PR[90,1] + -20.406;
   1:  PR[91,2] = PR[90,2] + -14.558;
   1:  PR[91,3] = PR[90,3] + 52.996;
   1:L PR[91] R[100]mm/sec CNT100;
   1:  PR[91,1] = PR[90,1] + -19.605;
   1:  PR[91,2] = PR[90,2] + -15.342;
   1:  PR[91,3] = PR[90,3] + 53.006;
   1:L PR[91] R[100]mm/sec CNT100;
   1:  PR[91,1] = PR[90,1] + -18.762;
   1:  PR[91,2] = PR[90,2] + -16.085;
   1:  PR[91,3] = PR[90,3] + 53.016;
   1:L PR[91] R[100]mm/sec CNT100;
   1:  PR[91,1] = PR[90,1] + -17.881;
   1:  PR[91,2] = PR[90,2] + -16.787;
   1:  PR[91,3] = PR[90,3] + 53.025;
   1:L PR[91] R[100]mm/sec CNT100;
   1:  PR[91,1] = PR[90,1] + -16.965;
   1:  PR[91,2] = PR[90,2] + -17.444;
   1:  PR[91,3] = PR[90,3] + 53.035;
   1:L PR[91] R[100]mm/sec CNT100;
   1:  PR[91,1] = PR[90,1] + -16.014;
   1:  PR[91,2] = PR[90,2] + -18.055;
   1:  PR[91,3] = PR[90,3] + 53.045;
   1:L PR[91] R[100]mm/sec CNT100;
   1:  PR[91,1] = PR[90,1] + -15.032;
   1:  PR[91,2] = PR[90,2] + -18.619;
   1:  PR[91,3] = PR[90,3] + 53.054;
   1:L PR[91] R[100]mm/sec CNT100;
   1:  PR[91,1] = PR[90,1] + -14.021;
   1:  PR[91,2] = PR[90,2] + -19.134;
   1:  PR[91,3] = PR[90,3] + 53.064;
   1:L PR[91] R[100]mm/sec CNT100;
   1:  PR[91,1] = PR[90,1] + -12.984;
   1:  PR[91,2] = PR[90,2] + -19.598;
   1:  PR[91,3] = PR[90,3] + 53.074;
   1:L PR[91] R[100]mm/sec CNT100;
   1:  PR[91,1] = PR[90,1] + -11.923;
   1:  PR[91,2] = PR[90,2] + -20.009;
   1:  PR[91,3] = PR[90,3] + 53.083;
   1:L PR[91] R[100]mm/sec CNT100;
   1:  PR[91,1] = PR[90,1] + -10.842;
   1:  PR[91,2] = PR[90,2] + -20.367;
   1:  PR[91,3] = PR[90,3] + 53.093;
   1:L PR[91] R[100]mm/sec CNT100;
   1:  PR[91,1] = PR[90,1] + -9.742;
   1:  PR[91,2] = PR[90,2] + -20.671;
   1:  PR[91,3] = PR[90,3] + 53.103;
   1:L PR[91] R[100]mm/sec CNT100;
   1:  PR[91,1] = PR[90,1] + -8.627;
   1:  PR[91,2] = PR[90,2] + -20.919;
   1:  PR[91,3] = PR[90,3] + 53.113;
   1:L PR[91] R[100]mm/sec CNT100;
   1:  PR[91,1] = PR[90,1] + -7.500;
   1:  PR[91,2] = PR[90,2] + -21.111;
   1:  PR[91,3] = PR[90,3] + 53.123;
   1:L PR[91] R[100]mm/sec CNT100;
   1:  PR[91,1] = PR[90,1] + -6.364;
   1:  PR[91,2] = PR[90,2] + -21.245;
   1:  PR[91,3] = PR[90,3] + 53.132;
   1:L PR[91] R[100]mm/sec CNT100;
   1:  PR[91,1] = PR[90,1] + -5.221;
   1:  PR[91,2] = PR[90,2] + -21.322;
   1:  PR[91,3] = PR[90,3] + 53.142;
   1:L PR[91] R[100]mm/sec CNT100;
   1:  PR[91,1] = PR[90,1] + -4.076;
   1:  PR[91,2] = PR[90,2] + -21.341;
   1:  PR[91,3] = PR[90,3] + 53.152;
   1:L PR[91] R[100]mm/sec CNT100;
   1:  PR[91,1] = PR[90,1] + -2.930;
   1:  PR[91,2] = PR[90,2] + -21.302;
   1:  PR[91,3] = PR[90,3] + 53.162;
   1:L PR[91] R[100]mm/sec CNT100;
   1:  PR[91,1] = PR[90,1] + -1.788;
   1:  PR[91,2] = PR[90,2] + -21.205;
   1:  PR[91,3] = PR[90,3] + 53.172;
   1:L PR[91] R[100]mm/sec CNT100;
   1:  PR[91,1] = PR[90,1] + -0.576;
   1:  PR[91,2] = PR[90,2] + -21.038;
   1:  PR[91,3] = PR[90,3] + 53.182;
   1:L PR[91] R[100]mm/sec CNT100;
   1:  PR[91,1] = PR[90,1] + -0.120;
   1:  PR[91,2] = PR[90,2] + -21.001;
   1:  PR[91,3] = PR[90,3] + 53.192;
   1:L PR[91] R[100]mm/sec CNT100;
   1:  PR[91,1] = PR[90,1] + 0.347;
   1:  PR[91,2] = PR[90,2] + -21.040;
   1:  PR[91,3] = PR[90,3] + 53.196;
   1:L PR[91] R[100]mm/sec CNT100;
   1:  PR[91] = PR[90];
   1:  PR[91,1] = PR[90,1] + 0.963;
   1:  PR[91,2] = PR[90,2] + -21.475;
   1:  PR[91,3] = PR[90,3] + 54.530;
   1:L PR[91] R[100]mm/sec CNT100;
   1:  PR[91,1] = PR[90,1] + 2.124;
   1:  PR[91,2] = PR[90,2] + -21.576;
   1:  PR[91,3] = PR[90,3] + 53.206;
   1:L PR[91] R[100]mm/sec CNT100;
   1:  PR[91,1] = PR[90,1] + 3.284;
   1:  PR[91,2] = PR[90,2] + -21.618;
   1:  PR[91,3] = PR[90,3] + 53.216;
   1:L PR[91] R[100]mm/sec CNT100;
   1:  PR[91,1] = PR[90,1] + 4.443;
   1:  PR[91,2] = PR[90,2] + -21.601;
   1:  PR[91,3] = PR[90,3] + 53.226;
   1:L PR[91] R[100]mm/sec CNT100;
   1:  PR[91,1] = PR[90,1] + 5.599;
   1:  PR[91,2] = PR[90,2] + -21.525;
   1:  PR[91,3] = PR[90,3] + 53.236;
   1:L PR[91] R[100]mm/sec CNT100;
   1:  PR[91,1] = PR[90,1] + 6.750;
   1:  PR[91,2] = PR[90,2] + -21.391;
   1:  PR[91,3] = PR[90,3] + 53.246;
   1:L PR[91] R[100]mm/sec CNT100;
   1:  PR[91,1] = PR[90,1] + 7.888;
   1:  PR[91,2] = PR[90,2] + -21.199;
   1:  PR[91,3] = PR[90,3] + 53.256;
   1:L PR[91] R[100]mm/sec CNT100;
   1:  PR[91,1] = PR[90,1] + 9.260;
   1:  PR[91,2] = PR[90,2] + -20.884;
   1:  PR[91,3] = PR[90,3] + 53.266;
   1:L PR[91] R[100]mm/sec CNT100;
   1:  PR[91,1] = PR[90,1] + 10.132;
   1:  PR[91,2] = PR[90,2] + -20.643;
   1:  PR[91,3] = PR[90,3] + 53.278;
   1:L PR[91] R[100]mm/sec CNT100;
   1:  PR[91,1] = PR[90,1] + 11.227;
   1:  PR[91,2] = PR[90,2] + -20.281;
   1:  PR[91,3] = PR[90,3] + 53.286;
   1:L PR[91] R[100]mm/sec CNT100;
   1:  PR[91,1] = PR[90,1] + 12.301;
   1:  PR[91,2] = PR[90,2] + -19.865;
   1:  PR[91,3] = PR[90,3] + 53.296;
   1:L PR[91] R[100]mm/sec CNT100;
   1:  PR[91,1] = PR[90,1] + 13.351;
   1:  PR[91,2] = PR[90,2] + -19.396;
   1:  PR[91,3] = PR[90,3] + 53.305;
   1:L PR[91] R[100]mm/sec CNT100;
   1:  PR[91,1] = PR[90,1] + 14.375;
   1:  PR[91,2] = PR[90,2] + -18.876;
   1:  PR[91,3] = PR[90,3] + 53.315;
   1:L PR[91] R[100]mm/sec CNT100;
   1:  PR[91,1] = PR[90,1] + 15.369;
   1:  PR[91,2] = PR[90,2] + -18.305;
   1:  PR[91,3] = PR[90,3] + 53.325;
   1:L PR[91] R[100]mm/sec CNT100;
   1:  PR[91,1] = PR[90,1] + 16.331;
   1:  PR[91,2] = PR[90,2] + -17.686;
   1:  PR[91,3] = PR[90,3] + 53.335;
   1:L PR[91] R[100]mm/sec CNT100;
   1:  PR[91,1] = PR[90,1] + 17.263;
   1:  PR[91,2] = PR[90,2] + -17.017;
   1:  PR[91,3] = PR[90,3] + 53.345;
   1:L PR[91] R[100]mm/sec CNT100;
   1:  PR[91,1] = PR[90,1] + 18.150;
   1:  PR[91,2] = PR[90,2] + -16.310;
   1:  PR[91,3] = PR[90,3] + 53.355;
   1:L PR[91] R[100]mm/sec CNT100;
   1:  PR[91,1] = PR[90,1] + 19.003;
   1:  PR[91,2] = PR[90,2] + -15.558;
   1:  PR[91,3] = PR[90,3] + 53.365;
   1:L PR[91] R[100]mm/sec CNT100;
   1:  PR[91,1] = PR[90,1] + 19.815;
   1:  PR[91,2] = PR[90,2] + -14.764;
   1:  PR[91,3] = PR[90,3] + 53.374;
   1:L PR[91] R[100]mm/sec CNT100;
   1:  PR[91,1] = PR[90,1] + 20.584;
   1:  PR[91,2] = PR[90,2] + -13.932;
   1:  PR[91,3] = PR[90,3] + 53.384;
   1:L PR[91] R[100]mm/sec CNT100;
   1:  PR[91,1] = PR[90,1] + 21.308;
   1:  PR[91,2] = PR[90,2] + -13.062;
   1:  PR[91,3] = PR[90,3] + 53.394;
   1:L PR[91] R[100]mm/sec CNT100;
   1:  PR[91,1] = PR[90,1] + 21.986;
   1:  PR[91,2] = PR[90,2] + -12.158;
   1:  PR[91,3] = PR[90,3] + 53.404;
   1:L PR[91] R[100]mm/sec CNT100;
   1:  PR[91,1] = PR[90,1] + 22.616;
   1:  PR[91,2] = PR[90,2] + -11.221;
   1:  PR[91,3] = PR[90,3] + 53.413;
   1:L PR[91] R[100]mm/sec CNT100;
   1:  PR[91,1] = PR[90,1] + 23.197;
   1:  PR[91,2] = PR[90,2] + -10.256;
   1:  PR[91,3] = PR[90,3] + 53.423;
   1:L PR[91] R[100]mm/sec CNT100;
   1:  PR[91,1] = PR[90,1] + 23.726;
   1:  PR[91,2] = PR[90,2] + -9.264;
   1:  PR[91,3] = PR[90,3] + 53.433;
   1:L PR[91] R[100]mm/sec CNT100;
   1:  PR[91,1] = PR[90,1] + 24.203;
   1:  PR[91,2] = PR[90,2] + -8.250;
   1:  PR[91,3] = PR[90,3] + 53.442;
   1:L PR[91] R[100]mm/sec CNT100;
   1:  PR[91,1] = PR[90,1] + 24.627;
   1:  PR[91,2] = PR[90,2] + -7.215;
   1:  PR[91,3] = PR[90,3] + 53.452;
   1:L PR[91] R[100]mm/sec CNT100;
   1:  PR[91,1] = PR[90,1] + 24.996;
   1:  PR[91,2] = PR[90,2] + -6.163;
   1:  PR[91,3] = PR[90,3] + 53.462;
   1:L PR[91] R[100]mm/sec CNT100;
   1:  PR[91,1] = PR[90,1] + 25.309;
   1:  PR[91,2] = PR[90,2] + -5.096;
   1:  PR[91,3] = PR[90,3] + 53.471;
   1:L PR[91] R[100]mm/sec CNT100;
   1:  PR[91,1] = PR[90,1] + 25.567;
   1:  PR[91,2] = PR[90,2] + -4.015;
   1:  PR[91,3] = PR[90,3] + 53.481;
   1:L PR[91] R[100]mm/sec CNT100;
   1:  PR[91,1] = PR[90,1] + 25.768;
   1:  PR[91,2] = PR[90,2] + -2.921;
   1:  PR[91,3] = PR[90,3] + 53.490;
   1:L PR[91] R[100]mm/sec CNT100;
   1:  PR[91,1] = PR[90,1] + 25.912;
   1:  PR[91,2] = PR[90,2] + -1.815;
   1:  PR[91,3] = PR[90,3] + 53.500;
   1:L PR[91] R[100]mm/sec CNT100;
   1:  PR[91,1] = PR[90,1] + 25.999;
   1:  PR[91,2] = PR[90,2] + -0.699;
   1:  PR[91,3] = PR[90,3] + 53.510;
   1:L PR[91] R[100]mm/sec CNT100;
   1:  PR[91,1] = PR[90,1] + 26.027;
   1:  PR[91,2] = PR[90,2] + 0.428;
   1:  PR[91,3] = PR[90,3] + 53.519;
   1:L PR[91] R[100]mm/sec CNT100;
   1:  PR[91,1] = PR[90,1] + 25.999;
   1:  PR[91,2] = PR[90,2] + 1.554;
   1:  PR[91,3] = PR[90,3] + 53.529;
   1:L PR[91] R[100]mm/sec CNT100;
   1:  PR[91,1] = PR[90,1] + 25.912;
   1:  PR[91,2] = PR[90,2] + 2.670;
   1:  PR[91,3] = PR[90,3] + 53.539;
   1:L PR[91] R[100]mm/sec CNT100;
   1:  PR[91,1] = PR[90,1] + 25.768;
   1:  PR[91,2] = PR[90,2] + 3.776;
   1:  PR[91,3] = PR[90,3] + 53.548;
   1:L PR[91] R[100]mm/sec CNT100;
   1:  PR[91,1] = PR[90,1] + 25.567;
   1:  PR[91,2] = PR[90,2] + 4.869;
   1:  PR[91,3] = PR[90,3] + 53.558;
   1:L PR[91] R[100]mm/sec CNT100;
   1:  PR[91,1] = PR[90,1] + 25.310;
   1:  PR[91,2] = PR[90,2] + 5.951;
   1:  PR[91,3] = PR[90,3] + 53.567;
   1:L PR[91] R[100]mm/sec CNT100;
   1:  PR[91,1] = PR[90,1] + 24.996;
   1:  PR[91,2] = PR[90,2] + 7.018;
   1:  PR[91,3] = PR[90,3] + 53.577;
   1:L PR[91] R[100]mm/sec CNT100;
   1:  PR[91,1] = PR[90,1] + 24.627;
   1:  PR[91,2] = PR[90,2] + 8.069;
   1:  PR[91,3] = PR[90,3] + 53.587;
   1:L PR[91] R[100]mm/sec CNT100;
   1:  PR[91,1] = PR[90,1] + 24.203;
   1:  PR[91,2] = PR[90,2] + 9.104;
   1:  PR[91,3] = PR[90,3] + 53.596;
   1:L PR[91] R[100]mm/sec CNT100;
   1:  PR[91,1] = PR[90,1] + 23.727;
   1:  PR[91,2] = PR[90,2] + 10.118;
   1:  PR[91,3] = PR[90,3] + 53.606;
   1:L PR[91] R[100]mm/sec CNT100;
   1:  PR[91,1] = PR[90,1] + 23.197;
   1:  PR[91,2] = PR[90,2] + 11.110;
   1:  PR[91,3] = PR[90,3] + 53.615;
   1:L PR[91] R[100]mm/sec CNT100;
   1:  PR[91,1] = PR[90,1] + 22.617;
   1:  PR[91,2] = PR[90,2] + 12.075;
   1:  PR[91,3] = PR[90,3] + 53.625;
   1:L PR[91] R[100]mm/sec CNT100;
   1:  PR[91,1] = PR[90,1] + 21.987;
   1:  PR[91,2] = PR[90,2] + 13.011;
   1:  PR[91,3] = PR[90,3] + 53.635;
   1:L PR[91] R[100]mm/sec CNT100;
   1:  PR[91,1] = PR[90,1] + 21.310;
   1:  PR[91,2] = PR[90,2] + 13.916;
   1:  PR[91,3] = PR[90,3] + 53.645;
   1:L PR[91] R[100]mm/sec CNT100;
   1:  PR[91,1] = PR[90,1] + 20.585;
   1:  PR[91,2] = PR[90,2] + 14.785;
   1:  PR[91,3] = PR[90,3] + 53.654;
   1:L PR[91] R[100]mm/sec CNT100;
   1:  PR[91,1] = PR[90,1] + 19.817;
   1:  PR[91,2] = PR[90,2] + 15.618;
   1:  PR[91,3] = PR[90,3] + 53.664;
   1:L PR[91] R[100]mm/sec CNT100;
   1:  PR[91,1] = PR[90,1] + 19.005;
   1:  PR[91,2] = PR[90,2] + 16.411;
   1:  PR[91,3] = PR[90,3] + 53.674;
   1:L PR[91] R[100]mm/sec CNT100;
   1:  PR[91,1] = PR[90,1] + 18.153;
   1:  PR[91,2] = PR[90,2] + 17.164;
   1:  PR[91,3] = PR[90,3] + 53.684;
   1:L PR[91] R[100]mm/sec CNT100;
   1:  PR[91,1] = PR[90,1] + 17.261;
   1:  PR[91,2] = PR[90,2] + 17.874;
   1:  PR[91,3] = PR[90,3] + 53.693;
   1:L PR[91] R[100]mm/sec CNT100;
   1:  PR[91,1] = PR[90,1] + 16.333;
   1:  PR[91,2] = PR[90,2] + 18.539;
   1:  PR[91,3] = PR[90,3] + 53.703;
   1:L PR[91] R[100]mm/sec CNT100;
   1:  PR[91,1] = PR[90,1] + 15.372;
   1:  PR[91,2] = PR[90,2] + 19.158;
   1:  PR[91,3] = PR[90,3] + 53.713;
   1:L PR[91] R[100]mm/sec CNT100;
   1:  PR[91,1] = PR[90,1] + 14.378;
   1:  PR[91,2] = PR[90,2] + 19.729;
   1:  PR[91,3] = PR[90,3] + 53.723;
   1:L PR[91] R[100]mm/sec CNT100;
   1:  PR[91,1] = PR[90,1] + 13.354;
   1:  PR[91,2] = PR[90,2] + 20.250;
   1:  PR[91,3] = PR[90,3] + 53.733;
   1:L PR[91] R[100]mm/sec CNT100;
   1:  PR[91,1] = PR[90,1] + 12.305;
   1:  PR[91,2] = PR[90,2] + 20.719;
   1:  PR[91,3] = PR[90,3] + 53.743;
   1:L PR[91] R[100]mm/sec CNT100;
   1:  PR[91,1] = PR[90,1] + 11.231;
   1:  PR[91,2] = PR[90,2] + 21.135;
   1:  PR[91,3] = PR[90,3] + 53.752;
   1:L PR[91] R[100]mm/sec CNT100;
   1:  PR[91,1] = PR[90,1] + 10.136;
   1:  PR[91,2] = PR[90,2] + 21.497;
   1:  PR[91,3] = PR[90,3] + 53.762;
   1:L PR[91] R[100]mm/sec CNT100;
   1:  PR[91,1] = PR[90,1] + 9.023;
   1:  PR[91,2] = PR[90,2] + 21.803;
   1:  PR[91,3] = PR[90,3] + 53.772;
   1:L PR[91] R[100]mm/sec CNT100;
   1:  PR[91,1] = PR[90,1] + 7.895;
   1:  PR[91,2] = PR[90,2] + 22.053;
   1:  PR[91,3] = PR[90,3] + 53.782;
   1:L PR[91] R[100]mm/sec CNT100;
   1:  PR[91,1] = PR[90,1] + 6.755;
   1:  PR[91,2] = PR[90,2] + 22.245;
   1:  PR[91,3] = PR[90,3] + 53.792;
   1:L PR[91] R[100]mm/sec CNT100;
   1:  PR[91,1] = PR[90,1] + 5.605;
   1:  PR[91,2] = PR[90,2] + 22.380;
   1:  PR[91,3] = PR[90,3] + 53.802;
   1:L PR[91] R[100]mm/sec CNT100;
   1:  PR[91,1] = PR[90,1] + 4.448;
   1:  PR[91,2] = PR[90,2] + 22.456;
   1:  PR[91,3] = PR[90,3] + 53.812;
   1:L PR[91] R[100]mm/sec CNT100;
   1:  PR[91,1] = PR[90,1] + 3.686;
   1:  PR[91,2] = PR[90,2] + 22.469;
   1:  PR[91,3] = PR[90,3] + 53.822;
   1:L PR[91] R[100]mm/sec CNT100;
   1:  PR[91,1] = PR[90,1] + 3.290;
   1:  PR[91,2] = PR[90,2] + 22.474;
   1:  PR[91,3] = PR[90,3] + 53.829;
   1:L PR[91] R[100]mm/sec CNT100;
   1:  PR[91,1] = PR[90,1] + 2.130;
   1:  PR[91,2] = PR[90,2] + 22.432;
   1:  PR[91,3] = PR[90,3] + 53.832;
   1:L PR[91] R[100]mm/sec CNT100;
   1:  PR[91,1] = PR[90,1] + 0.971;
   1:  PR[91,2] = PR[90,2] + 22.331;
   1:  PR[91,3] = PR[90,3] + 53.842;
   1:L PR[91] R[100]mm/sec CNT100;
   1:  PR[91,1] = PR[90,1] + 0.288;
   1:  PR[91,2] = PR[90,2] + 22.239;
   1:  PR[91,3] = PR[90,3] + 53.852;
   1:L PR[91] R[100]mm/sec CNT100;
   1:  PR[91,1] = PR[90,1] + -0.065;
   1:  PR[91,2] = PR[90,2] + 22.210;
   1:  PR[91,3] = PR[90,3] + 53.858;
   1:L PR[91] R[100]mm/sec CNT100;
   1:  PR[91,1] = PR[90,1] + -0.520;
   1:  PR[91,2] = PR[90,2] + 22.239;
   1:  PR[91,3] = PR[90,3] + 53.861;
   1:L PR[91] R[100]mm/sec CNT100;
   1:  PR[91,1] = PR[90,1] + -1.210;
   1:  PR[91,2] = PR[90,2] + 22.331;
   1:  PR[91,3] = PR[90,3] + 53.865;
   1:L PR[91] R[100]mm/sec CNT100;
   1:  PR[91,1] = PR[90,1] + -2.368;
   1:  PR[91,2] = PR[90,2] + 22.432;
   1:  PR[91,3] = PR[90,3] + 53.871;
   1:L PR[91] R[100]mm/sec CNT100;
   1:  PR[91,1] = PR[90,1] + -3.527;
   1:  PR[91,2] = PR[90,2] + 22.473;
   1:  PR[91,3] = PR[90,3] + 53.881;
   1:L PR[91] R[100]mm/sec CNT100;
   1:  PR[91,1] = PR[90,1] + -4.687;
   1:  PR[91,2] = PR[90,2] + 22.456;
   1:  PR[91,3] = PR[90,3] + 53.891;
   1:L PR[91] R[100]mm/sec CNT100;
   1:  PR[91,1] = PR[90,1] + -5.843;
   1:  PR[91,2] = PR[90,2] + 22.380;
   1:  PR[91,3] = PR[90,3] + 53.901;
   1:L PR[91] R[100]mm/sec CNT100;
   1:  PR[91,1] = PR[90,1] + -6.993;
   1:  PR[91,2] = PR[90,2] + 22.245;
   1:  PR[91,3] = PR[90,3] + 53.911;
   1:L PR[91] R[100]mm/sec CNT100;
   1:  PR[91,1] = PR[90,1] + -8.131;
   1:  PR[91,2] = PR[90,2] + 22.053;
   1:  PR[91,3] = PR[90,3] + 53.921;
   1:L PR[91] R[100]mm/sec CNT100;
   1:  PR[91,1] = PR[90,1] + -9.503;
   1:  PR[91,2] = PR[90,2] + 21.738;
   1:  PR[91,3] = PR[90,3] + 53.931;
   1:L PR[91] R[100]mm/sec CNT100;
   1:  PR[91,1] = PR[90,1] + -10.374;
   1:  PR[91,2] = PR[90,2] + 21.497;
   1:  PR[91,3] = PR[90,3] + 53.943;
   1:L PR[91] R[100]mm/sec CNT100;
   1:  PR[91,1] = PR[90,1] + -11.469;
   1:  PR[91,2] = PR[90,2] + 21.135;
   1:  PR[91,3] = PR[90,3] + 53.951;
   1:L PR[91] R[100]mm/sec CNT100;
   1:  PR[91,1] = PR[90,1] + -12.543;
   1:  PR[91,2] = PR[90,2] + 20.719;
   1:  PR[91,3] = PR[90,3] + 53.961;
   1:L PR[91] R[100]mm/sec CNT100;
   1:  PR[91,1] = PR[90,1] + -13.593;
   1:  PR[91,2] = PR[90,2] + 20.250;
   1:  PR[91,3] = PR[90,3] + 53.971;
   1:L PR[91] R[100]mm/sec CNT100;
   1:  PR[91,1] = PR[90,1] + -14.616;
   1:  PR[91,2] = PR[90,2] + 19.729;
   1:  PR[91,3] = PR[90,3] + 53.980;
   1:L PR[91] R[100]mm/sec CNT100;
   1:  PR[91,1] = PR[90,1] + -15.610;
   1:  PR[91,2] = PR[90,2] + 19.158;
   1:  PR[91,3] = PR[90,3] + 53.990;
   1:L PR[91] R[100]mm/sec CNT100;
   1:  PR[91,1] = PR[90,1] + -16.572;
   1:  PR[91,2] = PR[90,2] + 18.539;
   1:  PR[91,3] = PR[90,3] + 54.000;
   1:L PR[91] R[100]mm/sec CNT100;
   1:  PR[91,1] = PR[90,1] + -17.504;
   1:  PR[91,2] = PR[90,2] + 17.870;
   1:  PR[91,3] = PR[90,3] + 54.010;
   1:L PR[91] R[100]mm/sec CNT100;
   1:  PR[91,1] = PR[90,1] + -18.391;
   1:  PR[91,2] = PR[90,2] + 17.163;
   1:  PR[91,3] = PR[90,3] + 54.020;
   1:L PR[91] R[100]mm/sec CNT100;
   1:  PR[91,1] = PR[90,1] + -19.243;
   1:  PR[91,2] = PR[90,2] + 16.411;
   1:  PR[91,3] = PR[90,3] + 54.030;
   1:L PR[91] R[100]mm/sec CNT100;
   1:  PR[91,1] = PR[90,1] + -20.055;
   1:  PR[91,2] = PR[90,2] + 15.618;
   1:  PR[91,3] = PR[90,3] + 54.039;
   1:L PR[91] R[100]mm/sec CNT100;
   1:  PR[91,1] = PR[90,1] + -20.824;
   1:  PR[91,2] = PR[90,2] + 14.786;
   1:  PR[91,3] = PR[90,3] + 54.049;
   1:L PR[91] R[100]mm/sec CNT100;
   1:  PR[91,1] = PR[90,1] + -21.548;
   1:  PR[91,2] = PR[90,2] + 13.917;
   1:  PR[91,3] = PR[90,3] + 54.059;
   1:L PR[91] R[100]mm/sec CNT100;
   1:  PR[91,1] = PR[90,1] + -22.226;
   1:  PR[91,2] = PR[90,2] + 13.013;
   1:  PR[91,3] = PR[90,3] + 54.069;
   1:L PR[91] R[100]mm/sec CNT100;
   1:  PR[91,1] = PR[90,1] + -22.855;
   1:  PR[91,2] = PR[90,2] + 12.077;
   1:  PR[91,3] = PR[90,3] + 54.078;
   1:L PR[91] R[100]mm/sec CNT100;
   1:  PR[91,1] = PR[90,1] + -23.436;
   1:  PR[91,2] = PR[90,2] + 11.112;
   1:  PR[91,3] = PR[90,3] + 54.088;
   1:L PR[91] R[100]mm/sec CNT100;
   1:  PR[91,1] = PR[90,1] + -23.965;
   1:  PR[91,2] = PR[90,2] + 10.119;
   1:  PR[91,3] = PR[90,3] + 54.098;
   1:L PR[91] R[100]mm/sec CNT100;
   1:  PR[91,1] = PR[90,1] + -24.442;
   1:  PR[91,2] = PR[90,2] + 9.104;
   1:  PR[91,3] = PR[90,3] + 54.107;
   1:L PR[91] R[100]mm/sec CNT100;
   1:  PR[91,1] = PR[90,1] + -24.865;
   1:  PR[91,2] = PR[90,2] + 8.068;
   1:  PR[91,3] = PR[90,3] + 54.117;
   1:L PR[91] R[100]mm/sec CNT100;
   1:  PR[91,1] = PR[90,1] + -25.234;
   1:  PR[91,2] = PR[90,2] + 7.015;
   1:  PR[91,3] = PR[90,3] + 54.127;
   1:L PR[91] R[100]mm/sec CNT100;
   1:  PR[91,1] = PR[90,1] + -25.548;
   1:  PR[91,2] = PR[90,2] + 5.947;
   1:  PR[91,3] = PR[90,3] + 54.136;
   1:L PR[91] R[100]mm/sec CNT100;
   1:  PR[91,1] = PR[90,1] + -25.806;
   1:  PR[91,2] = PR[90,2] + 4.866;
   1:  PR[91,3] = PR[90,3] + 54.146;
   1:L PR[91] R[100]mm/sec CNT100;
   1:  PR[91,1] = PR[90,1] + -26.007;
   1:  PR[91,2] = PR[90,2] + 3.773;
   1:  PR[91,3] = PR[90,3] + 54.156;
   1:L PR[91] R[100]mm/sec CNT100;
   1:  PR[91,1] = PR[90,1] + -26.151;
   1:  PR[91,2] = PR[90,2] + 2.669;
   1:  PR[91,3] = PR[90,3] + 54.165;
   1:L PR[91] R[100]mm/sec CNT100;
   1:  PR[91,1] = PR[90,1] + -26.237;
   1:  PR[91,2] = PR[90,2] + 1.553;
   1:  PR[91,3] = PR[90,3] + 54.175;
   1:L PR[91] R[100]mm/sec CNT100;
   1:  PR[91,1] = PR[90,1] + -26.265;
   1:  PR[91,2] = PR[90,2] + 0.428;
   1:  PR[91,3] = PR[90,3] + 54.184;
   1:L PR[91] R[100]mm/sec CNT100;
   1:  PR[91,1] = PR[90,1] + -26.237;
   1:  PR[91,2] = PR[90,2] + -0.698;
   1:  PR[91,3] = PR[90,3] + 54.194;
   1:L PR[91] R[100]mm/sec CNT100;
   1:  PR[91,1] = PR[90,1] + -26.150;
   1:  PR[91,2] = PR[90,2] + -1.814;
   1:  PR[91,3] = PR[90,3] + 54.204;
   1:L PR[91] R[100]mm/sec CNT100;
   1:  PR[91,1] = PR[90,1] + -26.007;
   1:  PR[91,2] = PR[90,2] + -2.918;
   1:  PR[91,3] = PR[90,3] + 54.213;
   1:L PR[91] R[100]mm/sec CNT100;
   1:  PR[91,1] = PR[90,1] + -25.805;
   1:  PR[91,2] = PR[90,2] + -4.012;
   1:  PR[91,3] = PR[90,3] + 54.223;
   1:L PR[91] R[100]mm/sec CNT100;
   1:  PR[91,1] = PR[90,1] + -25.548;
   1:  PR[91,2] = PR[90,2] + -5.093;
   1:  PR[91,3] = PR[90,3] + 54.232;
   1:L PR[91] R[100]mm/sec CNT100;
   1:  PR[91,1] = PR[90,1] + -25.234;
   1:  PR[91,2] = PR[90,2] + -6.161;
   1:  PR[91,3] = PR[90,3] + 54.242;
   1:L PR[91] R[100]mm/sec CNT100;
   1:  PR[91,1] = PR[90,1] + -24.865;
   1:  PR[91,2] = PR[90,2] + -7.214;
   1:  PR[91,3] = PR[90,3] + 54.252;
   1:L PR[91] R[100]mm/sec CNT100;
   1:  PR[91,1] = PR[90,1] + -24.441;
   1:  PR[91,2] = PR[90,2] + -8.250;
   1:  PR[91,3] = PR[90,3] + 54.261;
   1:L PR[91] R[100]mm/sec CNT100;
   1:  PR[91,1] = PR[90,1] + -23.964;
   1:  PR[91,2] = PR[90,2] + -9.265;
   1:  PR[91,3] = PR[90,3] + 54.271;
   1:L PR[91] R[100]mm/sec CNT100;
   1:  PR[91,1] = PR[90,1] + -23.435;
   1:  PR[91,2] = PR[90,2] + -10.258;
   1:  PR[91,3] = PR[90,3] + 54.281;
   1:L PR[91] R[100]mm/sec CNT100;
   1:  PR[91,1] = PR[90,1] + -22.855;
   1:  PR[91,2] = PR[90,2] + -11.224;
   1:  PR[91,3] = PR[90,3] + 54.290;
   1:L PR[91] R[100]mm/sec CNT100;
   1:  PR[91,1] = PR[90,1] + -22.225;
   1:  PR[91,2] = PR[90,2] + -12.160;
   1:  PR[91,3] = PR[90,3] + 54.300;
   1:L PR[91] R[100]mm/sec CNT100;
   1:  PR[91,1] = PR[90,1] + -21.547;
   1:  PR[91,2] = PR[90,2] + -13.063;
   1:  PR[91,3] = PR[90,3] + 54.310;
   1:L PR[91] R[100]mm/sec CNT100;
   1:  PR[91,1] = PR[90,1] + -20.822;
   1:  PR[91,2] = PR[90,2] + -13.932;
   1:  PR[91,3] = PR[90,3] + 54.319;
   1:L PR[91] R[100]mm/sec CNT100;
   1:  PR[91,1] = PR[90,1] + -20.053;
   1:  PR[91,2] = PR[90,2] + -14.765;
   1:  PR[91,3] = PR[90,3] + 54.329;
   1:L PR[91] R[100]mm/sec CNT100;
   1:  PR[91,1] = PR[90,1] + -19.241;
   1:  PR[91,2] = PR[90,2] + -15.558;
   1:  PR[91,3] = PR[90,3] + 54.339;
   1:L PR[91] R[100]mm/sec CNT100;
   1:  PR[91,1] = PR[90,1] + -18.389;
   1:  PR[91,2] = PR[90,2] + -16.310;
   1:  PR[91,3] = PR[90,3] + 54.349;
   1:L PR[91] R[100]mm/sec CNT100;
   1:  PR[91,1] = PR[90,1] + -17.497;
   1:  PR[91,2] = PR[90,2] + -17.020;
   1:  PR[91,3] = PR[90,3] + 54.358;
   1:L PR[91] R[100]mm/sec CNT100;
   1:  PR[91,1] = PR[90,1] + -16.569;
   1:  PR[91,2] = PR[90,2] + -17.686;
   1:  PR[91,3] = PR[90,3] + 54.368;
   1:L PR[91] R[100]mm/sec CNT100;
   1:  PR[91,1] = PR[90,1] + -15.607;
   1:  PR[91,2] = PR[90,2] + -18.305;
   1:  PR[91,3] = PR[90,3] + 54.378;
   1:L PR[91] R[100]mm/sec CNT100;
   1:  PR[91,1] = PR[90,1] + -14.613;
   1:  PR[91,2] = PR[90,2] + -18.876;
   1:  PR[91,3] = PR[90,3] + 54.388;
   1:L PR[91] R[100]mm/sec CNT100;
   1:  PR[91,1] = PR[90,1] + -13.589;
   1:  PR[91,2] = PR[90,2] + -19.396;
   1:  PR[91,3] = PR[90,3] + 54.398;
   1:L PR[91] R[100]mm/sec CNT100;
   1:  PR[91,1] = PR[90,1] + -12.539;
   1:  PR[91,2] = PR[90,2] + -19.865;
   1:  PR[91,3] = PR[90,3] + 54.408;
   1:L PR[91] R[100]mm/sec CNT100;
   1:  PR[91,1] = PR[90,1] + -11.466;
   1:  PR[91,2] = PR[90,2] + -20.281;
   1:  PR[91,3] = PR[90,3] + 54.417;
   1:L PR[91] R[100]mm/sec CNT100;
   1:  PR[91,1] = PR[90,1] + -10.370;
   1:  PR[91,2] = PR[90,2] + -20.643;
   1:  PR[91,3] = PR[90,3] + 54.427;
   1:L PR[91] R[100]mm/sec CNT100;
   1:  PR[91,1] = PR[90,1] + -9.257;
   1:  PR[91,2] = PR[90,2] + -20.949;
   1:  PR[91,3] = PR[90,3] + 54.437;
   1:L PR[91] R[100]mm/sec CNT100;
   1:  PR[91,1] = PR[90,1] + -8.129;
   1:  PR[91,2] = PR[90,2] + -21.199;
   1:  PR[91,3] = PR[90,3] + 54.447;
   1:L PR[91] R[100]mm/sec CNT100;
   1:  PR[91,1] = PR[90,1] + -6.988;
   1:  PR[91,2] = PR[90,2] + -21.391;
   1:  PR[91,3] = PR[90,3] + 54.457;
   1:L PR[91] R[100]mm/sec CNT100;
   1:  PR[91,1] = PR[90,1] + -5.838;
   1:  PR[91,2] = PR[90,2] + -21.525;
   1:  PR[91,3] = PR[90,3] + 54.467;
   1:L PR[91] R[100]mm/sec CNT100;
   1:  PR[91,1] = PR[90,1] + -4.681;
   1:  PR[91,2] = PR[90,2] + -21.601;
   1:  PR[91,3] = PR[90,3] + 54.477;
   1:L PR[91] R[100]mm/sec CNT100;
   1:  PR[91,1] = PR[90,1] + -3.919;
   1:  PR[91,2] = PR[90,2] + -21.614;
   1:  PR[91,3] = PR[90,3] + 54.487;
   1:L PR[91] R[100]mm/sec CNT100;
   1:  PR[91,1] = PR[90,1] + -3.523;
   1:  PR[91,2] = PR[90,2] + -21.618;
   1:  PR[91,3] = PR[90,3] + 54.494;
   1:L PR[91] R[100]mm/sec CNT100;
   1:  PR[91,1] = PR[90,1] + -2.362;
   1:  PR[91,2] = PR[90,2] + -21.576;
   1:  PR[91,3] = PR[90,3] + 54.497;
   1:L PR[91] R[100]mm/sec CNT100;
   1:  PR[91,1] = PR[90,1] + -1.202;
   1:  PR[91,2] = PR[90,2] + -21.475;
   1:  PR[91,3] = PR[90,3] + 54.507;
   1:L PR[91] R[100]mm/sec CNT100;
   1:  PR[91,1] = PR[90,1] + -0.520;
   1:  PR[91,2] = PR[90,2] + -21.383;
   1:  PR[91,3] = PR[90,3] + 54.517;
   1:L PR[91] R[100]mm/sec CNT100;
   1:  PR[91,1] = PR[90,1] + -0.065;
   1:  PR[91,2] = PR[90,2] + -21.355;
   1:  PR[91,3] = PR[90,3] + 54.523;
   1:L PR[91] R[100]mm/sec CNT100;
   1:  PR[91,1] = PR[90,1] + 0.288;
   1:  PR[91,2] = PR[90,2] + -21.384;
   1:  PR[91,3] = PR[90,3] + 54.527;
   1:L PR[91] R[100]mm/sec CNT100;
   1:  PR[91] = PR[90];
   1:  PR[91,1] = PR[90,1] + 1.551;
   1:  PR[91,2] = PR[90,2] + -21.853;
   1:  PR[91,3] = PR[90,3] + 55.860;
   1:L PR[91] R[100]mm/sec CNT100;
   1:  PR[91,1] = PR[90,1] + 2.722;
   1:  PR[91,2] = PR[90,2] + -21.900;
   1:  PR[91,3] = PR[90,3] + 54.544;
   1:L PR[91] R[100]mm/sec CNT100;
   1:  PR[91,1] = PR[90,1] + 3.894;
   1:  PR[91,2] = PR[90,2] + -21.886;
   1:  PR[91,3] = PR[90,3] + 54.554;
   1:L PR[91] R[100]mm/sec CNT100;
   1:  PR[91,1] = PR[90,1] + 5.064;
   1:  PR[91,2] = PR[90,2] + -21.813;
   1:  PR[91,3] = PR[90,3] + 54.564;
   1:L PR[91] R[100]mm/sec CNT100;
   1:  PR[91,1] = PR[90,1] + 5.964;
   1:  PR[91,2] = PR[90,2] + -21.712;
   1:  PR[91,3] = PR[90,3] + 54.574;
   1:L PR[91] R[100]mm/sec CNT100;
   1:  PR[91,1] = PR[90,1] + 6.226;
   1:  PR[91,2] = PR[90,2] + -21.681;
   1:  PR[91,3] = PR[90,3] + 54.582;
   1:L PR[91] R[100]mm/sec CNT100;
   1:  PR[91,1] = PR[90,1] + 7.381;
   1:  PR[91,2] = PR[90,2] + -21.489;
   1:  PR[91,3] = PR[90,3] + 54.584;
   1:L PR[91] R[100]mm/sec CNT100;
   1:  PR[91,1] = PR[90,1] + 8.524;
   1:  PR[91,2] = PR[90,2] + -21.240;
   1:  PR[91,3] = PR[90,3] + 54.594;
   1:L PR[91] R[100]mm/sec CNT100;
   1:  PR[91,1] = PR[90,1] + 9.316;
   1:  PR[91,2] = PR[90,2] + -21.025;
   1:  PR[91,3] = PR[90,3] + 54.604;
   1:L PR[91] R[100]mm/sec CNT100;
   1:  PR[91,1] = PR[90,1] + 9.649;
   1:  PR[91,2] = PR[90,2] + -20.933;
   1:  PR[91,3] = PR[90,3] + 54.611;
   1:L PR[91] R[100]mm/sec CNT100;
   1:  PR[91,1] = PR[90,1] + 10.759;
   1:  PR[91,2] = PR[90,2] + -20.570;
   1:  PR[91,3] = PR[90,3] + 54.614;
   1:L PR[91] R[100]mm/sec CNT100;
   1:  PR[91,1] = PR[90,1] + 11.847;
   1:  PR[91,2] = PR[90,2] + -20.151;
   1:  PR[91,3] = PR[90,3] + 54.624;
   1:L PR[91] R[100]mm/sec CNT100;
   1:  PR[91,1] = PR[90,1] + 12.520;
   1:  PR[91,2] = PR[90,2] + -19.853;
   1:  PR[91,3] = PR[90,3] + 54.634;
   1:L PR[91] R[100]mm/sec CNT100;
   1:  PR[91,1] = PR[90,1] + 12.909;
   1:  PR[91,2] = PR[90,2] + -19.679;
   1:  PR[91,3] = PR[90,3] + 54.641;
   1:L PR[91] R[100]mm/sec CNT100;
   1:  PR[91,1] = PR[90,1] + 13.947;
   1:  PR[91,2] = PR[90,2] + -19.154;
   1:  PR[91,3] = PR[90,3] + 54.644;
   1:L PR[91] R[100]mm/sec CNT100;
   1:  PR[91,1] = PR[90,1] + 14.954;
   1:  PR[91,2] = PR[90,2] + -18.578;
   1:  PR[91,3] = PR[90,3] + 54.654;
   1:L PR[91] R[100]mm/sec CNT100;
   1:  PR[91,1] = PR[90,1] + 15.929;
   1:  PR[91,2] = PR[90,2] + -17.952;
   1:  PR[91,3] = PR[90,3] + 54.664;
   1:L PR[91] R[100]mm/sec CNT100;
   1:  PR[91,1] = PR[90,1] + 16.870;
   1:  PR[91,2] = PR[90,2] + -17.279;
   1:  PR[91,3] = PR[90,3] + 54.674;
   1:L PR[91] R[100]mm/sec CNT100;
   1:  PR[91,1] = PR[90,1] + 17.774;
   1:  PR[91,2] = PR[90,2] + -16.560;
   1:  PR[91,3] = PR[90,3] + 54.684;
   1:L PR[91] R[100]mm/sec CNT100;
   1:  PR[91,1] = PR[90,1] + 18.639;
   1:  PR[91,2] = PR[90,2] + -15.798;
   1:  PR[91,3] = PR[90,3] + 54.694;
   1:L PR[91] R[100]mm/sec CNT100;
   1:  PR[91,1] = PR[90,1] + 19.463;
   1:  PR[91,2] = PR[90,2] + -14.993;
   1:  PR[91,3] = PR[90,3] + 54.704;
   1:L PR[91] R[100]mm/sec CNT100;
   1:  PR[91,1] = PR[90,1] + 20.243;
   1:  PR[91,2] = PR[90,2] + -14.149;
   1:  PR[91,3] = PR[90,3] + 54.714;
   1:L PR[91] R[100]mm/sec CNT100;
   1:  PR[91,1] = PR[90,1] + 20.978;
   1:  PR[91,2] = PR[90,2] + -13.267;
   1:  PR[91,3] = PR[90,3] + 54.724;
   1:L PR[91] R[100]mm/sec CNT100;
   1:  PR[91,1] = PR[90,1] + 21.665;
   1:  PR[91,2] = PR[90,2] + -12.349;
   1:  PR[91,3] = PR[90,3] + 54.734;
   1:L PR[91] R[100]mm/sec CNT100;
   1:  PR[91,1] = PR[90,1] + 22.304;
   1:  PR[91,2] = PR[90,2] + -11.400;
   1:  PR[91,3] = PR[90,3] + 54.744;
   1:L PR[91] R[100]mm/sec CNT100;
   1:  PR[91,1] = PR[90,1] + 22.893;
   1:  PR[91,2] = PR[90,2] + -10.420;
   1:  PR[91,3] = PR[90,3] + 54.754;
   1:L PR[91] R[100]mm/sec CNT100;
   1:  PR[91,1] = PR[90,1] + 23.430;
   1:  PR[91,2] = PR[90,2] + -9.414;
   1:  PR[91,3] = PR[90,3] + 54.764;
   1:L PR[91] R[100]mm/sec CNT100;
   1:  PR[91,1] = PR[90,1] + 23.914;
   1:  PR[91,2] = PR[90,2] + -8.384;
   1:  PR[91,3] = PR[90,3] + 54.773;
   1:L PR[91] R[100]mm/sec CNT100;
   1:  PR[91,1] = PR[90,1] + 24.344;
   1:  PR[91,2] = PR[90,2] + -7.333;
   1:  PR[91,3] = PR[90,3] + 54.783;
   1:L PR[91] R[100]mm/sec CNT100;
   1:  PR[91,1] = PR[90,1] + 24.718;
   1:  PR[91,2] = PR[90,2] + -6.264;
   1:  PR[91,3] = PR[90,3] + 54.793;
   1:L PR[91] R[100]mm/sec CNT100;
   1:  PR[91,1] = PR[90,1] + 25.036;
   1:  PR[91,2] = PR[90,2] + -5.179;
   1:  PR[91,3] = PR[90,3] + 54.803;
   1:L PR[91] R[100]mm/sec CNT100;
   1:  PR[91,1] = PR[90,1] + 25.298;
   1:  PR[91,2] = PR[90,2] + -4.080;
   1:  PR[91,3] = PR[90,3] + 54.813;
   1:L PR[91] R[100]mm/sec CNT100;
   1:  PR[91,1] = PR[90,1] + 25.501;
   1:  PR[91,2] = PR[90,2] + -2.969;
   1:  PR[91,3] = PR[90,3] + 54.822;
   1:L PR[91] R[100]mm/sec CNT100;
   1:  PR[91,1] = PR[90,1] + 25.647;
   1:  PR[91,2] = PR[90,2] + -1.846;
   1:  PR[91,3] = PR[90,3] + 54.832;
   1:L PR[91] R[100]mm/sec CNT100;
   1:  PR[91,1] = PR[90,1] + 25.735;
   1:  PR[91,2] = PR[90,2] + -0.713;
   1:  PR[91,3] = PR[90,3] + 54.842;
   1:L PR[91] R[100]mm/sec CNT100;
   1:  PR[91,1] = PR[90,1] + 25.763;
   1:  PR[91,2] = PR[90,2] + 0.428;
   1:  PR[91,3] = PR[90,3] + 54.852;
   1:L PR[91] R[100]mm/sec CNT100;
   1:  PR[91,1] = PR[90,1] + 25.735;
   1:  PR[91,2] = PR[90,2] + 1.568;
   1:  PR[91,3] = PR[90,3] + 54.862;
   1:L PR[91] R[100]mm/sec CNT100;
   1:  PR[91,1] = PR[90,1] + 25.647;
   1:  PR[91,2] = PR[90,2] + 2.701;
   1:  PR[91,3] = PR[90,3] + 54.871;
   1:L PR[91] R[100]mm/sec CNT100;
   1:  PR[91,1] = PR[90,1] + 25.502;
   1:  PR[91,2] = PR[90,2] + 3.823;
   1:  PR[91,3] = PR[90,3] + 54.881;
   1:L PR[91] R[100]mm/sec CNT100;
   1:  PR[91,1] = PR[90,1] + 25.298;
   1:  PR[91,2] = PR[90,2] + 4.935;
   1:  PR[91,3] = PR[90,3] + 54.891;
   1:L PR[91] R[100]mm/sec CNT100;
   1:  PR[91,1] = PR[90,1] + 25.036;
   1:  PR[91,2] = PR[90,2] + 6.034;
   1:  PR[91,3] = PR[90,3] + 54.901;
   1:L PR[91] R[100]mm/sec CNT100;
   1:  PR[91,1] = PR[90,1] + 24.718;
   1:  PR[91,2] = PR[90,2] + 7.118;
   1:  PR[91,3] = PR[90,3] + 54.910;
   1:L PR[91] R[100]mm/sec CNT100;
   1:  PR[91,1] = PR[90,1] + 24.344;
   1:  PR[91,2] = PR[90,2] + 8.187;
   1:  PR[91,3] = PR[90,3] + 54.920;
   1:L PR[91] R[100]mm/sec CNT100;
   1:  PR[91,1] = PR[90,1] + 23.914;
   1:  PR[91,2] = PR[90,2] + 9.238;
   1:  PR[91,3] = PR[90,3] + 54.930;
   1:L PR[91] R[100]mm/sec CNT100;
   1:  PR[91,1] = PR[90,1] + 23.431;
   1:  PR[91,2] = PR[90,2] + 10.268;
   1:  PR[91,3] = PR[90,3] + 54.940;
   1:L PR[91] R[100]mm/sec CNT100;
   1:  PR[91,1] = PR[90,1] + 22.894;
   1:  PR[91,2] = PR[90,2] + 11.274;
   1:  PR[91,3] = PR[90,3] + 54.950;
   1:L PR[91] R[100]mm/sec CNT100;
   1:  PR[91,1] = PR[90,1] + 22.305;
   1:  PR[91,2] = PR[90,2] + 12.253;
   1:  PR[91,3] = PR[90,3] + 54.959;
   1:L PR[91] R[100]mm/sec CNT100;
   1:  PR[91,1] = PR[90,1] + 21.667;
   1:  PR[91,2] = PR[90,2] + 13.203;
   1:  PR[91,3] = PR[90,3] + 54.969;
   1:L PR[91] R[100]mm/sec CNT100;
   1:  PR[91,1] = PR[90,1] + 20.979;
   1:  PR[91,2] = PR[90,2] + 14.120;
   1:  PR[91,3] = PR[90,3] + 54.979;
   1:L PR[91] R[100]mm/sec CNT100;
   1:  PR[91,1] = PR[90,1] + 20.244;
   1:  PR[91,2] = PR[90,2] + 15.002;
   1:  PR[91,3] = PR[90,3] + 54.989;
   1:L PR[91] R[100]mm/sec CNT100;
   1:  PR[91,1] = PR[90,1] + 19.465;
   1:  PR[91,2] = PR[90,2] + 15.846;
   1:  PR[91,3] = PR[90,3] + 54.999;
   1:L PR[91] R[100]mm/sec CNT100;
   1:  PR[91,1] = PR[90,1] + 18.641;
   1:  PR[91,2] = PR[90,2] + 16.651;
   1:  PR[91,3] = PR[90,3] + 55.009;
   1:L PR[91] R[100]mm/sec CNT100;
   1:  PR[91,1] = PR[90,1] + 17.777;
   1:  PR[91,2] = PR[90,2] + 17.414;
   1:  PR[91,3] = PR[90,3] + 55.019;
   1:L PR[91] R[100]mm/sec CNT100;
   1:  PR[91,1] = PR[90,1] + 16.873;
   1:  PR[91,2] = PR[90,2] + 18.133;
   1:  PR[91,3] = PR[90,3] + 55.029;
   1:L PR[91] R[100]mm/sec CNT100;
   1:  PR[91,1] = PR[90,1] + 15.932;
   1:  PR[91,2] = PR[90,2] + 18.805;
   1:  PR[91,3] = PR[90,3] + 55.039;
   1:L PR[91] R[100]mm/sec CNT100;
   1:  PR[91,1] = PR[90,1] + 14.957;
   1:  PR[91,2] = PR[90,2] + 19.431;
   1:  PR[91,3] = PR[90,3] + 55.049;
   1:L PR[91] R[100]mm/sec CNT100;
   1:  PR[91,1] = PR[90,1] + 13.950;
   1:  PR[91,2] = PR[90,2] + 20.007;
   1:  PR[91,3] = PR[90,3] + 55.059;
   1:L PR[91] R[100]mm/sec CNT100;
   1:  PR[91,1] = PR[90,1] + 12.913;
   1:  PR[91,2] = PR[90,2] + 20.532;
   1:  PR[91,3] = PR[90,3] + 55.069;
   1:L PR[91] R[100]mm/sec CNT100;
   1:  PR[91,1] = PR[90,1] + 11.850;
   1:  PR[91,2] = PR[90,2] + 21.005;
   1:  PR[91,3] = PR[90,3] + 55.079;
   1:L PR[91] R[100]mm/sec CNT100;
   1:  PR[91,1] = PR[90,1] + 10.763;
   1:  PR[91,2] = PR[90,2] + 21.423;
   1:  PR[91,3] = PR[90,3] + 55.089;
   1:L PR[91] R[100]mm/sec CNT100;
   1:  PR[91,1] = PR[90,1] + 9.655;
   1:  PR[91,2] = PR[90,2] + 21.787;
   1:  PR[91,3] = PR[90,3] + 55.099;
   1:L PR[91] R[100]mm/sec CNT100;
   1:  PR[91,1] = PR[90,1] + 8.528;
   1:  PR[91,2] = PR[90,2] + 22.094;
   1:  PR[91,3] = PR[90,3] + 55.109;
   1:L PR[91] R[100]mm/sec CNT100;
   1:  PR[91,1] = PR[90,1] + 7.385;
   1:  PR[91,2] = PR[90,2] + 22.344;
   1:  PR[91,3] = PR[90,3] + 55.119;
   1:L PR[91] R[100]mm/sec CNT100;
   1:  PR[91,1] = PR[90,1] + 7.099;
   1:  PR[91,2] = PR[90,2] + 22.393;
   1:  PR[91,3] = PR[90,3] + 55.129;
   1:L PR[91] R[100]mm/sec CNT100;
   1:  PR[91,1] = PR[90,1] + 6.233;
   1:  PR[91,2] = PR[90,2] + 22.535;
   1:  PR[91,3] = PR[90,3] + 55.132;
   1:L PR[91] R[100]mm/sec CNT100;
   1:  PR[91,1] = PR[90,1] + 5.069;
   1:  PR[91,2] = PR[90,2] + 22.668;
   1:  PR[91,3] = PR[90,3] + 55.139;
   1:L PR[91] R[100]mm/sec CNT100;
   1:  PR[91,1] = PR[90,1] + 3.900;
   1:  PR[91,2] = PR[90,2] + 22.741;
   1:  PR[91,3] = PR[90,3] + 55.149;
   1:L PR[91] R[100]mm/sec CNT100;
   1:  PR[91,1] = PR[90,1] + 2.728;
   1:  PR[91,2] = PR[90,2] + 22.755;
   1:  PR[91,3] = PR[90,3] + 55.159;
   1:L PR[91] R[100]mm/sec CNT100;
   1:  PR[91,1] = PR[90,1] + 1.557;
   1:  PR[91,2] = PR[90,2] + 22.709;
   1:  PR[91,3] = PR[90,3] + 55.169;
   1:L PR[91] R[100]mm/sec CNT100;
   1:  PR[91,1] = PR[90,1] + -0.007;
   1:  PR[91,2] = PR[90,2] + 22.562;
   1:  PR[91,3] = PR[90,3] + 55.180;
   1:L PR[91] R[100]mm/sec CNT100;
   1:  PR[91,1] = PR[90,1] + -0.455;
   1:  PR[91,2] = PR[90,2] + 22.581;
   1:  PR[91,3] = PR[90,3] + 55.193;
   1:L PR[91] R[100]mm/sec CNT100;
   1:  PR[91,1] = PR[90,1] + -1.796;
   1:  PR[91,2] = PR[90,2] + 22.709;
   1:  PR[91,3] = PR[90,3] + 55.197;
   1:L PR[91] R[100]mm/sec CNT100;
   1:  PR[91,1] = PR[90,1] + -2.967;
   1:  PR[91,2] = PR[90,2] + 22.755;
   1:  PR[91,3] = PR[90,3] + 55.209;
   1:L PR[91] R[100]mm/sec CNT100;
   1:  PR[91,1] = PR[90,1] + -4.139;
   1:  PR[91,2] = PR[90,2] + 22.741;
   1:  PR[91,3] = PR[90,3] + 55.219;
   1:L PR[91] R[100]mm/sec CNT100;
   1:  PR[91,1] = PR[90,1] + -5.308;
   1:  PR[91,2] = PR[90,2] + 22.668;
   1:  PR[91,3] = PR[90,3] + 55.229;
   1:L PR[91] R[100]mm/sec CNT100;
   1:  PR[91,1] = PR[90,1] + -6.471;
   1:  PR[91,2] = PR[90,2] + 22.535;
   1:  PR[91,3] = PR[90,3] + 55.239;
   1:L PR[91] R[100]mm/sec CNT100;
   1:  PR[91,1] = PR[90,1] + -7.625;
   1:  PR[91,2] = PR[90,2] + 22.343;
   1:  PR[91,3] = PR[90,3] + 55.249;
   1:L PR[91] R[100]mm/sec CNT100;
   1:  PR[91,1] = PR[90,1] + -8.456;
   1:  PR[91,2] = PR[90,2] + 22.163;
   1:  PR[91,3] = PR[90,3] + 55.259;
   1:L PR[91] R[100]mm/sec CNT100;
   1:  PR[91,1] = PR[90,1] + -8.765;
   1:  PR[91,2] = PR[90,2] + 22.094;
   1:  PR[91,3] = PR[90,3] + 55.266;
   1:L PR[91] R[100]mm/sec CNT100;
   1:  PR[91,1] = PR[90,1] + -9.893;
   1:  PR[91,2] = PR[90,2] + 21.787;
   1:  PR[91,3] = PR[90,3] + 55.269;
   1:L PR[91] R[100]mm/sec CNT100;
   1:  PR[91,1] = PR[90,1] + -11.001;
   1:  PR[91,2] = PR[90,2] + 21.424;
   1:  PR[91,3] = PR[90,3] + 55.279;
   1:L PR[91] R[100]mm/sec CNT100;
   1:  PR[91,1] = PR[90,1] + -12.089;
   1:  PR[91,2] = PR[90,2] + 21.005;
   1:  PR[91,3] = PR[90,3] + 55.289;
   1:L PR[91] R[100]mm/sec CNT100;
   1:  PR[91,1] = PR[90,1] + -13.152;
   1:  PR[91,2] = PR[90,2] + 20.532;
   1:  PR[91,3] = PR[90,3] + 55.299;
   1:L PR[91] R[100]mm/sec CNT100;
   1:  PR[91,1] = PR[90,1] + -14.188;
   1:  PR[91,2] = PR[90,2] + 20.007;
   1:  PR[91,3] = PR[90,3] + 55.309;
   1:L PR[91] R[100]mm/sec CNT100;
   1:  PR[91,1] = PR[90,1] + -15.196;
   1:  PR[91,2] = PR[90,2] + 19.431;
   1:  PR[91,3] = PR[90,3] + 55.319;
   1:L PR[91] R[100]mm/sec CNT100;
   1:  PR[91,1] = PR[90,1] + -16.171;
   1:  PR[91,2] = PR[90,2] + 18.805;
   1:  PR[91,3] = PR[90,3] + 55.329;
   1:L PR[91] R[100]mm/sec CNT100;
   1:  PR[91,1] = PR[90,1] + -17.111;
   1:  PR[91,2] = PR[90,2] + 18.132;
   1:  PR[91,3] = PR[90,3] + 55.339;
   1:L PR[91] R[100]mm/sec CNT100;
   1:  PR[91,1] = PR[90,1] + -18.015;
   1:  PR[91,2] = PR[90,2] + 17.413;
   1:  PR[91,3] = PR[90,3] + 55.349;
   1:L PR[91] R[100]mm/sec CNT100;
   1:  PR[91,1] = PR[90,1] + -18.880;
   1:  PR[91,2] = PR[90,2] + 16.651;
   1:  PR[91,3] = PR[90,3] + 55.359;
   1:L PR[91] R[100]mm/sec CNT100;
   1:  PR[91,1] = PR[90,1] + -19.703;
   1:  PR[91,2] = PR[90,2] + 15.846;
   1:  PR[91,3] = PR[90,3] + 55.369;
   1:L PR[91] R[100]mm/sec CNT100;
   1:  PR[91,1] = PR[90,1] + -20.483;
   1:  PR[91,2] = PR[90,2] + 15.002;
   1:  PR[91,3] = PR[90,3] + 55.379;
   1:L PR[91] R[100]mm/sec CNT100;
   1:  PR[91,1] = PR[90,1] + -21.218;
   1:  PR[91,2] = PR[90,2] + 14.121;
   1:  PR[91,3] = PR[90,3] + 55.389;
   1:L PR[91] R[100]mm/sec CNT100;
   1:  PR[91,1] = PR[90,1] + -21.905;
   1:  PR[91,2] = PR[90,2] + 13.204;
   1:  PR[91,3] = PR[90,3] + 55.399;
   1:L PR[91] R[100]mm/sec CNT100;
   1:  PR[91,1] = PR[90,1] + -22.544;
   1:  PR[91,2] = PR[90,2] + 12.255;
   1:  PR[91,3] = PR[90,3] + 55.409;
   1:L PR[91] R[100]mm/sec CNT100;
   1:  PR[91,1] = PR[90,1] + -23.132;
   1:  PR[91,2] = PR[90,2] + 11.275;
   1:  PR[91,3] = PR[90,3] + 55.419;
   1:L PR[91] R[100]mm/sec CNT100;
   1:  PR[91,1] = PR[90,1] + -23.669;
   1:  PR[91,2] = PR[90,2] + 10.268;
   1:  PR[91,3] = PR[90,3] + 55.429;
   1:L PR[91] R[100]mm/sec CNT100;
   1:  PR[91,1] = PR[90,1] + -24.153;
   1:  PR[91,2] = PR[90,2] + 9.238;
   1:  PR[91,3] = PR[90,3] + 55.438;
   1:L PR[91] R[100]mm/sec CNT100;
   1:  PR[91,1] = PR[90,1] + -24.582;
   1:  PR[91,2] = PR[90,2] + 8.186;
   1:  PR[91,3] = PR[90,3] + 55.448;
   1:L PR[91] R[100]mm/sec CNT100;
   1:  PR[91,1] = PR[90,1] + -24.957;
   1:  PR[91,2] = PR[90,2] + 7.116;
   1:  PR[91,3] = PR[90,3] + 55.458;
   1:L PR[91] R[100]mm/sec CNT100;
   1:  PR[91,1] = PR[90,1] + -25.275;
   1:  PR[91,2] = PR[90,2] + 6.031;
   1:  PR[91,3] = PR[90,3] + 55.468;
   1:L PR[91] R[100]mm/sec CNT100;
   1:  PR[91,1] = PR[90,1] + -25.536;
   1:  PR[91,2] = PR[90,2] + 4.932;
   1:  PR[91,3] = PR[90,3] + 55.478;
   1:L PR[91] R[100]mm/sec CNT100;
   1:  PR[91,1] = PR[90,1] + -25.740;
   1:  PR[91,2] = PR[90,2] + 3.821;
   1:  PR[91,3] = PR[90,3] + 55.487;
   1:L PR[91] R[100]mm/sec CNT100;
   1:  PR[91,1] = PR[90,1] + -25.886;
   1:  PR[91,2] = PR[90,2] + 2.699;
   1:  PR[91,3] = PR[90,3] + 55.497;
   1:L PR[91] R[100]mm/sec CNT100;
   1:  PR[91,1] = PR[90,1] + -25.974;
   1:  PR[91,2] = PR[90,2] + 1.568;
   1:  PR[91,3] = PR[90,3] + 55.507;
   1:L PR[91] R[100]mm/sec CNT100;
   1:  PR[91,1] = PR[90,1] + -26.002;
   1:  PR[91,2] = PR[90,2] + 0.428;
   1:  PR[91,3] = PR[90,3] + 55.517;
   1:L PR[91] R[100]mm/sec CNT100;
   1:  PR[91,1] = PR[90,1] + -25.974;
   1:  PR[91,2] = PR[90,2] + -0.713;
   1:  PR[91,3] = PR[90,3] + 55.527;
   1:L PR[91] R[100]mm/sec CNT100;
   1:  PR[91,1] = PR[90,1] + -25.886;
   1:  PR[91,2] = PR[90,2] + -1.845;
   1:  PR[91,3] = PR[90,3] + 55.536;
   1:L PR[91] R[100]mm/sec CNT100;
   1:  PR[91,1] = PR[90,1] + -25.740;
   1:  PR[91,2] = PR[90,2] + -2.967;
   1:  PR[91,3] = PR[90,3] + 55.546;
   1:L PR[91] R[100]mm/sec CNT100;
   1:  PR[91,1] = PR[90,1] + -25.536;
   1:  PR[91,2] = PR[90,2] + -4.077;
   1:  PR[91,3] = PR[90,3] + 55.556;
   1:L PR[91] R[100]mm/sec CNT100;
   1:  PR[91,1] = PR[90,1] + -25.275;
   1:  PR[91,2] = PR[90,2] + -5.176;
   1:  PR[91,3] = PR[90,3] + 55.566;
   1:L PR[91] R[100]mm/sec CNT100;
   1:  PR[91,1] = PR[90,1] + -24.956;
   1:  PR[91,2] = PR[90,2] + -6.262;
   1:  PR[91,3] = PR[90,3] + 55.575;
   1:L PR[91] R[100]mm/sec CNT100;
   1:  PR[91,1] = PR[90,1] + -24.582;
   1:  PR[91,2] = PR[90,2] + -7.332;
   1:  PR[91,3] = PR[90,3] + 55.585;
   1:L PR[91] R[100]mm/sec CNT100;
   1:  PR[91,1] = PR[90,1] + -24.152;
   1:  PR[91,2] = PR[90,2] + -8.384;
   1:  PR[91,3] = PR[90,3] + 55.595;
   1:L PR[91] R[100]mm/sec CNT100;
   1:  PR[91,1] = PR[90,1] + -23.668;
   1:  PR[91,2] = PR[90,2] + -9.415;
   1:  PR[91,3] = PR[90,3] + 55.605;
   1:L PR[91] R[100]mm/sec CNT100;
   1:  PR[91,1] = PR[90,1] + -23.131;
   1:  PR[91,2] = PR[90,2] + -10.422;
   1:  PR[91,3] = PR[90,3] + 55.615;
   1:L PR[91] R[100]mm/sec CNT100;
   1:  PR[91,1] = PR[90,1] + -22.543;
   1:  PR[91,2] = PR[90,2] + -11.401;
   1:  PR[91,3] = PR[90,3] + 55.624;
   1:L PR[91] R[100]mm/sec CNT100;
   1:  PR[91,1] = PR[90,1] + -21.904;
   1:  PR[91,2] = PR[90,2] + -12.351;
   1:  PR[91,3] = PR[90,3] + 55.634;
   1:L PR[91] R[100]mm/sec CNT100;
   1:  PR[91,1] = PR[90,1] + -21.216;
   1:  PR[91,2] = PR[90,2] + -13.268;
   1:  PR[91,3] = PR[90,3] + 55.644;
   1:L PR[91] R[100]mm/sec CNT100;
   1:  PR[91,1] = PR[90,1] + -20.481;
   1:  PR[91,2] = PR[90,2] + -14.149;
   1:  PR[91,3] = PR[90,3] + 55.654;
   1:L PR[91] R[100]mm/sec CNT100;
   1:  PR[91,1] = PR[90,1] + -19.701;
   1:  PR[91,2] = PR[90,2] + -14.993;
   1:  PR[91,3] = PR[90,3] + 55.664;
   1:L PR[91] R[100]mm/sec CNT100;
   1:  PR[91,1] = PR[90,1] + -18.878;
   1:  PR[91,2] = PR[90,2] + -15.797;
   1:  PR[91,3] = PR[90,3] + 55.674;
   1:L PR[91] R[100]mm/sec CNT100;
   1:  PR[91,1] = PR[90,1] + -18.013;
   1:  PR[91,2] = PR[90,2] + -16.560;
   1:  PR[91,3] = PR[90,3] + 55.684;
   1:L PR[91] R[100]mm/sec CNT100;
   1:  PR[91,1] = PR[90,1] + -17.109;
   1:  PR[91,2] = PR[90,2] + -17.279;
   1:  PR[91,3] = PR[90,3] + 55.694;
   1:L PR[91] R[100]mm/sec CNT100;
   1:  PR[91,1] = PR[90,1] + -16.168;
   1:  PR[91,2] = PR[90,2] + -17.952;
   1:  PR[91,3] = PR[90,3] + 55.704;
   1:L PR[91] R[100]mm/sec CNT100;
   1:  PR[91,1] = PR[90,1] + -15.192;
   1:  PR[91,2] = PR[90,2] + -18.578;
   1:  PR[91,3] = PR[90,3] + 55.714;
   1:L PR[91] R[100]mm/sec CNT100;
   1:  PR[91,1] = PR[90,1] + -14.185;
   1:  PR[91,2] = PR[90,2] + -19.154;
   1:  PR[91,3] = PR[90,3] + 55.724;
   1:L PR[91] R[100]mm/sec CNT100;
   1:  PR[91,1] = PR[90,1] + -13.148;
   1:  PR[91,2] = PR[90,2] + -19.679;
   1:  PR[91,3] = PR[90,3] + 55.734;
   1:L PR[91] R[100]mm/sec CNT100;
   1:  PR[91,1] = PR[90,1] + -12.085;
   1:  PR[91,2] = PR[90,2] + -20.151;
   1:  PR[91,3] = PR[90,3] + 55.744;
   1:L PR[91] R[100]mm/sec CNT100;
   1:  PR[91,1] = PR[90,1] + -10.997;
   1:  PR[91,2] = PR[90,2] + -20.570;
   1:  PR[91,3] = PR[90,3] + 55.754;
   1:L PR[91] R[100]mm/sec CNT100;
   1:  PR[91,1] = PR[90,1] + -9.889;
   1:  PR[91,2] = PR[90,2] + -20.933;
   1:  PR[91,3] = PR[90,3] + 55.764;
   1:L PR[91] R[100]mm/sec CNT100;
   1:  PR[91,1] = PR[90,1] + -8.762;
   1:  PR[91,2] = PR[90,2] + -21.240;
   1:  PR[91,3] = PR[90,3] + 55.774;
   1:L PR[91] R[100]mm/sec CNT100;
   1:  PR[91,1] = PR[90,1] + -7.620;
   1:  PR[91,2] = PR[90,2] + -21.489;
   1:  PR[91,3] = PR[90,3] + 55.784;
   1:L PR[91] R[100]mm/sec CNT100;
   1:  PR[91,1] = PR[90,1] + -6.465;
   1:  PR[91,2] = PR[90,2] + -21.681;
   1:  PR[91,3] = PR[90,3] + 55.794;
   1:L PR[91] R[100]mm/sec CNT100;
   1:  PR[91,1] = PR[90,1] + -5.302;
   1:  PR[91,2] = PR[90,2] + -21.813;
   1:  PR[91,3] = PR[90,3] + 55.804;
   1:L PR[91] R[100]mm/sec CNT100;
   1:  PR[91,1] = PR[90,1] + -4.133;
   1:  PR[91,2] = PR[90,2] + -21.886;
   1:  PR[91,3] = PR[90,3] + 55.814;
   1:L PR[91] R[100]mm/sec CNT100;
   1:  PR[91,1] = PR[90,1] + -2.961;
   1:  PR[91,2] = PR[90,2] + -21.900;
   1:  PR[91,3] = PR[90,3] + 55.824;
   1:L PR[91] R[100]mm/sec CNT100;
   1:  PR[91,1] = PR[90,1] + -1.790;
   1:  PR[91,2] = PR[90,2] + -21.853;
   1:  PR[91,3] = PR[90,3] + 55.834;
   1:L PR[91] R[100]mm/sec CNT100;
   1:  PR[91,1] = PR[90,1] + -0.455;
   1:  PR[91,2] = PR[90,2] + -21.726;
   1:  PR[91,3] = PR[90,3] + 55.845;
   1:L PR[91] R[100]mm/sec CNT100;
   1:  PR[91,1] = PR[90,1] + -0.007;
   1:  PR[91,2] = PR[90,2] + -21.707;
   1:  PR[91,3] = PR[90,3] + 55.856;
   1:L PR[91] R[100]mm/sec CNT100;
   1:  PR[91] = PR[90];
   1:  PR[91,1] = PR[90,1] + 0.956;
   1:  PR[91,2] = PR[90,2] + -22.139;
   1:  PR[91,3] = PR[90,3] + 57.190;
   1:L PR[91] R[100]mm/sec CNT100;
   1:  PR[91,1] = PR[90,1] + 2.146;
   1:  PR[91,2] = PR[90,2] + -22.191;
   1:  PR[91,3] = PR[90,3] + 55.868;
   1:L PR[91] R[100]mm/sec CNT100;
   1:  PR[91,1] = PR[90,1] + 2.504;
   1:  PR[91,2] = PR[90,2] + -22.190;
   1:  PR[91,3] = PR[90,3] + 55.878;
   1:L PR[91] R[100]mm/sec CNT100;
   1:  PR[91,1] = PR[90,1] + 3.330;
   1:  PR[91,2] = PR[90,2] + -22.181;
   1:  PR[91,3] = PR[90,3] + 55.881;
   1:L PR[91] R[100]mm/sec CNT100;
   1:  PR[91,1] = PR[90,1] + 4.515;
   1:  PR[91,2] = PR[90,2] + -22.111;
   1:  PR[91,3] = PR[90,3] + 55.888;
   1:L PR[91] R[100]mm/sec CNT100;
   1:  PR[91,1] = PR[90,1] + 5.693;
   1:  PR[91,2] = PR[90,2] + -21.980;
   1:  PR[91,3] = PR[90,3] + 55.899;
   1:L PR[91] R[100]mm/sec CNT100;
   1:  PR[91,1] = PR[90,1] + 6.862;
   1:  PR[91,2] = PR[90,2] + -21.789;
   1:  PR[91,3] = PR[90,3] + 55.909;
   1:L PR[91] R[100]mm/sec CNT100;
   1:  PR[91,1] = PR[90,1] + 8.020;
   1:  PR[91,2] = PR[90,2] + -21.540;
   1:  PR[91,3] = PR[90,3] + 55.919;
   1:L PR[91] R[100]mm/sec CNT100;
   1:  PR[91,1] = PR[90,1] + 9.159;
   1:  PR[91,2] = PR[90,2] + -21.232;
   1:  PR[91,3] = PR[90,3] + 55.929;
   1:L PR[91] R[100]mm/sec CNT100;
   1:  PR[91,1] = PR[90,1] + 10.470;
   1:  PR[91,2] = PR[90,2] + -20.796;
   1:  PR[91,3] = PR[90,3] + 55.940;
   1:L PR[91] R[100]mm/sec CNT100;
   1:  PR[91,1] = PR[90,1] + 11.387;
   1:  PR[91,2] = PR[90,2] + -20.444;
   1:  PR[91,3] = PR[90,3] + 55.952;
   1:L PR[91] R[100]mm/sec CNT100;
   1:  PR[91,1] = PR[90,1] + 12.465;
   1:  PR[91,2] = PR[90,2] + -19.967;
   1:  PR[91,3] = PR[90,3] + 55.960;
   1:L PR[91] R[100]mm/sec CNT100;
   1:  PR[91,1] = PR[90,1] + 13.517;
   1:  PR[91,2] = PR[90,2] + -19.437;
   1:  PR[91,3] = PR[90,3] + 55.970;
   1:L PR[91] R[100]mm/sec CNT100;
   1:  PR[91,1] = PR[90,1] + 14.538;
   1:  PR[91,2] = PR[90,2] + -18.855;
   1:  PR[91,3] = PR[90,3] + 55.980;
   1:L PR[91] R[100]mm/sec CNT100;
   1:  PR[91,1] = PR[90,1] + 15.527;
   1:  PR[91,2] = PR[90,2] + -18.222;
   1:  PR[91,3] = PR[90,3] + 55.991;
   1:L PR[91] R[100]mm/sec CNT100;
   1:  PR[91,1] = PR[90,1] + 16.481;
   1:  PR[91,2] = PR[90,2] + -17.541;
   1:  PR[91,3] = PR[90,3] + 56.001;
   1:L PR[91] R[100]mm/sec CNT100;
   1:  PR[91,1] = PR[90,1] + 17.398;
   1:  PR[91,2] = PR[90,2] + -16.813;
   1:  PR[91,3] = PR[90,3] + 56.011;
   1:L PR[91] R[100]mm/sec CNT100;
   1:  PR[91,1] = PR[90,1] + 18.284;
   1:  PR[91,2] = PR[90,2] + -16.032;
   1:  PR[91,3] = PR[90,3] + 56.021;
   1:L PR[91] R[100]mm/sec CNT100;
   1:  PR[91,1] = PR[90,1] + 19.111;
   1:  PR[91,2] = PR[90,2] + -15.225;
   1:  PR[91,3] = PR[90,3] + 56.031;
   1:L PR[91] R[100]mm/sec CNT100;
   1:  PR[91,1] = PR[90,1] + 19.902;
   1:  PR[91,2] = PR[90,2] + -14.369;
   1:  PR[91,3] = PR[90,3] + 56.041;
   1:L PR[91] R[100]mm/sec CNT100;
   1:  PR[91,1] = PR[90,1] + 20.648;
   1:  PR[91,2] = PR[90,2] + -13.476;
   1:  PR[91,3] = PR[90,3] + 56.051;
   1:L PR[91] R[100]mm/sec CNT100;
   1:  PR[91,1] = PR[90,1] + 21.346;
   1:  PR[91,2] = PR[90,2] + -12.546;
   1:  PR[91,3] = PR[90,3] + 56.061;
   1:L PR[91] R[100]mm/sec CNT100;
   1:  PR[91,1] = PR[90,1] + 21.995;
   1:  PR[91,2] = PR[90,2] + -11.584;
   1:  PR[91,3] = PR[90,3] + 56.071;
   1:L PR[91] R[100]mm/sec CNT100;
   1:  PR[91,1] = PR[90,1] + 22.593;
   1:  PR[91,2] = PR[90,2] + -10.590;
   1:  PR[91,3] = PR[90,3] + 56.081;
   1:L PR[91] R[100]mm/sec CNT100;
   1:  PR[91,1] = PR[90,1] + 23.138;
   1:  PR[91,2] = PR[90,2] + -9.569;
   1:  PR[91,3] = PR[90,3] + 56.091;
   1:L PR[91] R[100]mm/sec CNT100;
   1:  PR[91,1] = PR[90,1] + 23.629;
   1:  PR[91,2] = PR[90,2] + -8.523;
   1:  PR[91,3] = PR[90,3] + 56.101;
   1:L PR[91] R[100]mm/sec CNT100;
   1:  PR[91,1] = PR[90,1] + 24.066;
   1:  PR[91,2] = PR[90,2] + -7.456;
   1:  PR[91,3] = PR[90,3] + 56.111;
   1:L PR[91] R[100]mm/sec CNT100;
   1:  PR[91,1] = PR[90,1] + 24.446;
   1:  PR[91,2] = PR[90,2] + -6.370;
   1:  PR[91,3] = PR[90,3] + 56.121;
   1:L PR[91] R[100]mm/sec CNT100;
   1:  PR[91,1] = PR[90,1] + 24.770;
   1:  PR[91,2] = PR[90,2] + -5.267;
   1:  PR[91,3] = PR[90,3] + 56.131;
   1:L PR[91] R[100]mm/sec CNT100;
   1:  PR[91,1] = PR[90,1] + 25.035;
   1:  PR[91,2] = PR[90,2] + -4.149;
   1:  PR[91,3] = PR[90,3] + 56.141;
   1:L PR[91] R[100]mm/sec CNT100;
   1:  PR[91,1] = PR[90,1] + 25.242;
   1:  PR[91,2] = PR[90,2] + -3.019;
   1:  PR[91,3] = PR[90,3] + 56.151;
   1:L PR[91] R[100]mm/sec CNT100;
   1:  PR[91,1] = PR[90,1] + 25.391;
   1:  PR[91,2] = PR[90,2] + -1.878;
   1:  PR[91,3] = PR[90,3] + 56.161;
   1:L PR[91] R[100]mm/sec CNT100;
   1:  PR[91,1] = PR[90,1] + 25.480;
   1:  PR[91,2] = PR[90,2] + -0.729;
   1:  PR[91,3] = PR[90,3] + 56.171;
   1:L PR[91] R[100]mm/sec CNT100;
   1:  PR[91,1] = PR[90,1] + 25.508;
   1:  PR[91,2] = PR[90,2] + 0.428;
   1:  PR[91,3] = PR[90,3] + 56.181;
   1:L PR[91] R[100]mm/sec CNT100;
   1:  PR[91,1] = PR[90,1] + 25.480;
   1:  PR[91,2] = PR[90,2] + 1.584;
   1:  PR[91,3] = PR[90,3] + 56.191;
   1:L PR[91] R[100]mm/sec CNT100;
   1:  PR[91,1] = PR[90,1] + 25.391;
   1:  PR[91,2] = PR[90,2] + 2.733;
   1:  PR[91,3] = PR[90,3] + 56.201;
   1:L PR[91] R[100]mm/sec CNT100;
   1:  PR[91,1] = PR[90,1] + 25.242;
   1:  PR[91,2] = PR[90,2] + 3.874;
   1:  PR[91,3] = PR[90,3] + 56.211;
   1:L PR[91] R[100]mm/sec CNT100;
   1:  PR[91,1] = PR[90,1] + 25.035;
   1:  PR[91,2] = PR[90,2] + 5.003;
   1:  PR[91,3] = PR[90,3] + 56.221;
   1:L PR[91] R[100]mm/sec CNT100;
   1:  PR[91,1] = PR[90,1] + 24.770;
   1:  PR[91,2] = PR[90,2] + 6.121;
   1:  PR[91,3] = PR[90,3] + 56.231;
   1:L PR[91] R[100]mm/sec CNT100;
   1:  PR[91,1] = PR[90,1] + 24.447;
   1:  PR[91,2] = PR[90,2] + 7.223;
   1:  PR[91,3] = PR[90,3] + 56.241;
   1:L PR[91] R[100]mm/sec CNT100;
   1:  PR[91,1] = PR[90,1] + 24.066;
   1:  PR[91,2] = PR[90,2] + 8.310;
   1:  PR[91,3] = PR[90,3] + 56.251;
   1:L PR[91] R[100]mm/sec CNT100;
   1:  PR[91,1] = PR[90,1] + 23.630;
   1:  PR[91,2] = PR[90,2] + 9.377;
   1:  PR[91,3] = PR[90,3] + 56.261;
   1:L PR[91] R[100]mm/sec CNT100;
   1:  PR[91,1] = PR[90,1] + 23.139;
   1:  PR[91,2] = PR[90,2] + 10.423;
   1:  PR[91,3] = PR[90,3] + 56.271;
   1:L PR[91] R[100]mm/sec CNT100;
   1:  PR[91,1] = PR[90,1] + 22.594;
   1:  PR[91,2] = PR[90,2] + 11.444;
   1:  PR[91,3] = PR[90,3] + 56.281;
   1:L PR[91] R[100]mm/sec CNT100;
   1:  PR[91,1] = PR[90,1] + 21.996;
   1:  PR[91,2] = PR[90,2] + 12.437;
   1:  PR[91,3] = PR[90,3] + 56.291;
   1:L PR[91] R[100]mm/sec CNT100;
   1:  PR[91,1] = PR[90,1] + 21.348;
   1:  PR[91,2] = PR[90,2] + 13.399;
   1:  PR[91,3] = PR[90,3] + 56.301;
   1:L PR[91] R[100]mm/sec CNT100;
   1:  PR[91,1] = PR[90,1] + 20.650;
   1:  PR[91,2] = PR[90,2] + 14.329;
   1:  PR[91,3] = PR[90,3] + 56.311;
   1:L PR[91] R[100]mm/sec CNT100;
   1:  PR[91,1] = PR[90,1] + 19.904;
   1:  PR[91,2] = PR[90,2] + 15.222;
   1:  PR[91,3] = PR[90,3] + 56.321;
   1:L PR[91] R[100]mm/sec CNT100;
   1:  PR[91,1] = PR[90,1] + 19.107;
   1:  PR[91,2] = PR[90,2] + 16.084;
   1:  PR[91,3] = PR[90,3] + 56.331;
   1:L PR[91] R[100]mm/sec CNT100;
   1:  PR[91,1] = PR[90,1] + 18.278;
   1:  PR[91,2] = PR[90,2] + 16.893;
   1:  PR[91,3] = PR[90,3] + 56.341;
   1:L PR[91] R[100]mm/sec CNT100;
   1:  PR[91,1] = PR[90,1] + 17.401;
   1:  PR[91,2] = PR[90,2] + 17.666;
   1:  PR[91,3] = PR[90,3] + 56.351;
   1:L PR[91] R[100]mm/sec CNT100;
   1:  PR[91,1] = PR[90,1] + 16.484;
   1:  PR[91,2] = PR[90,2] + 18.394;
   1:  PR[91,3] = PR[90,3] + 56.361;
   1:L PR[91] R[100]mm/sec CNT100;
   1:  PR[91,1] = PR[90,1] + 15.530;
   1:  PR[91,2] = PR[90,2] + 19.075;
   1:  PR[91,3] = PR[90,3] + 56.371;
   1:L PR[91] R[100]mm/sec CNT100;
   1:  PR[91,1] = PR[90,1] + 14.541;
   1:  PR[91,2] = PR[90,2] + 19.708;
   1:  PR[91,3] = PR[90,3] + 56.381;
   1:L PR[91] R[100]mm/sec CNT100;
   1:  PR[91,1] = PR[90,1] + 13.520;
   1:  PR[91,2] = PR[90,2] + 20.291;
   1:  PR[91,3] = PR[90,3] + 56.392;
   1:L PR[91] R[100]mm/sec CNT100;
   1:  PR[91,1] = PR[90,1] + 12.469;
   1:  PR[91,2] = PR[90,2] + 20.821;
   1:  PR[91,3] = PR[90,3] + 56.402;
   1:L PR[91] R[100]mm/sec CNT100;
   1:  PR[91,1] = PR[90,1] + 11.390;
   1:  PR[91,2] = PR[90,2] + 21.298;
   1:  PR[91,3] = PR[90,3] + 56.412;
   1:L PR[91] R[100]mm/sec CNT100;
   1:  PR[91,1] = PR[90,1] + 10.288;
   1:  PR[91,2] = PR[90,2] + 21.720;
   1:  PR[91,3] = PR[90,3] + 56.422;
   1:L PR[91] R[100]mm/sec CNT100;
   1:  PR[91,1] = PR[90,1] + 9.165;
   1:  PR[91,2] = PR[90,2] + 22.086;
   1:  PR[91,3] = PR[90,3] + 56.432;
   1:L PR[91] R[100]mm/sec CNT100;
   1:  PR[91,1] = PR[90,1] + 8.022;
   1:  PR[91,2] = PR[90,2] + 22.394;
   1:  PR[91,3] = PR[90,3] + 56.442;
   1:L PR[91] R[100]mm/sec CNT100;
   1:  PR[91,1] = PR[90,1] + 7.121;
   1:  PR[91,2] = PR[90,2] + 22.591;
   1:  PR[91,3] = PR[90,3] + 56.453;
   1:L PR[91] R[100]mm/sec CNT100;
   1:  PR[91,1] = PR[90,1] + 6.868;
   1:  PR[91,2] = PR[90,2] + 22.644;
   1:  PR[91,3] = PR[90,3] + 56.461;
   1:L PR[91] R[100]mm/sec CNT100;
   1:  PR[91,1] = PR[90,1] + 5.697;
   1:  PR[91,2] = PR[90,2] + 22.835;
   1:  PR[91,3] = PR[90,3] + 56.463;
   1:L PR[91] R[100]mm/sec CNT100;
   1:  PR[91,1] = PR[90,1] + 4.518;
   1:  PR[91,2] = PR[90,2] + 22.965;
   1:  PR[91,3] = PR[90,3] + 56.473;
   1:L PR[91] R[100]mm/sec CNT100;
   1:  PR[91,1] = PR[90,1] + 3.334;
   1:  PR[91,2] = PR[90,2] + 23.036;
   1:  PR[91,3] = PR[90,3] + 56.483;
   1:L PR[91] R[100]mm/sec CNT100;
   1:  PR[91,1] = PR[90,1] + 2.147;
   1:  PR[91,2] = PR[90,2] + 23.046;
   1:  PR[91,3] = PR[90,3] + 56.494;
   1:L PR[91] R[100]mm/sec CNT100;
   1:  PR[91,1] = PR[90,1] + 0.958;
   1:  PR[91,2] = PR[90,2] + 22.994;
   1:  PR[91,3] = PR[90,3] + 56.504;
   1:L PR[91] R[100]mm/sec CNT100;
   1:  PR[91,1] = PR[90,1] + 0.045;
   1:  PR[91,2] = PR[90,2] + 22.913;
   1:  PR[91,3] = PR[90,3] + 56.514;
   1:L PR[91] R[100]mm/sec CNT100;
   1:  PR[91,1] = PR[90,1] + -0.400;
   1:  PR[91,2] = PR[90,2] + 22.922;
   1:  PR[91,3] = PR[90,3] + 56.522;
   1:L PR[91] R[100]mm/sec CNT100;
   1:  PR[91,1] = PR[90,1] + -1.197;
   1:  PR[91,2] = PR[90,2] + 22.994;
   1:  PR[91,3] = PR[90,3] + 56.526;
   1:L PR[91] R[100]mm/sec CNT100;
   1:  PR[91,1] = PR[90,1] + -2.386;
   1:  PR[91,2] = PR[90,2] + 23.046;
   1:  PR[91,3] = PR[90,3] + 56.533;
   1:L PR[91] R[100]mm/sec CNT100;
   1:  PR[91,1] = PR[90,1] + -3.573;
   1:  PR[91,2] = PR[90,2] + 23.036;
   1:  PR[91,3] = PR[90,3] + 56.543;
   1:L PR[91] R[100]mm/sec CNT100;
   1:  PR[91,1] = PR[90,1] + -4.757;
   1:  PR[91,2] = PR[90,2] + 22.965;
   1:  PR[91,3] = PR[90,3] + 56.553;
   1:L PR[91] R[100]mm/sec CNT100;
   1:  PR[91,1] = PR[90,1] + -5.935;
   1:  PR[91,2] = PR[90,2] + 22.835;
   1:  PR[91,3] = PR[90,3] + 56.564;
   1:L PR[91] R[100]mm/sec CNT100;
   1:  PR[91,1] = PR[90,1] + -7.106;
   1:  PR[91,2] = PR[90,2] + 22.644;
   1:  PR[91,3] = PR[90,3] + 56.574;
   1:L PR[91] R[100]mm/sec CNT100;
   1:  PR[91,1] = PR[90,1] + -7.360;
   1:  PR[91,2] = PR[90,2] + 22.590;
   1:  PR[91,3] = PR[90,3] + 56.584;
   1:L PR[91] R[100]mm/sec CNT100;
   1:  PR[91,1] = PR[90,1] + -8.261;
   1:  PR[91,2] = PR[90,2] + 22.394;
   1:  PR[91,3] = PR[90,3] + 56.586;
   1:L PR[91] R[100]mm/sec CNT100;
   1:  PR[91,1] = PR[90,1] + -9.403;
   1:  PR[91,2] = PR[90,2] + 22.086;
   1:  PR[91,3] = PR[90,3] + 56.594;
   1:L PR[91] R[100]mm/sec CNT100;
   1:  PR[91,1] = PR[90,1] + -10.527;
   1:  PR[91,2] = PR[90,2] + 21.720;
   1:  PR[91,3] = PR[90,3] + 56.605;
   1:L PR[91] R[100]mm/sec CNT100;
   1:  PR[91,1] = PR[90,1] + -11.629;
   1:  PR[91,2] = PR[90,2] + 21.298;
   1:  PR[91,3] = PR[90,3] + 56.615;
   1:L PR[91] R[100]mm/sec CNT100;
   1:  PR[91,1] = PR[90,1] + -12.707;
   1:  PR[91,2] = PR[90,2] + 20.821;
   1:  PR[91,3] = PR[90,3] + 56.625;
   1:L PR[91] R[100]mm/sec CNT100;
   1:  PR[91,1] = PR[90,1] + -13.758;
   1:  PR[91,2] = PR[90,2] + 20.291;
   1:  PR[91,3] = PR[90,3] + 56.635;
   1:L PR[91] R[100]mm/sec CNT100;
   1:  PR[91,1] = PR[90,1] + -14.779;
   1:  PR[91,2] = PR[90,2] + 19.708;
   1:  PR[91,3] = PR[90,3] + 56.645;
   1:L PR[91] R[100]mm/sec CNT100;
   1:  PR[91,1] = PR[90,1] + -15.768;
   1:  PR[91,2] = PR[90,2] + 19.075;
   1:  PR[91,3] = PR[90,3] + 56.656;
   1:L PR[91] R[100]mm/sec CNT100;
   1:  PR[91,1] = PR[90,1] + -16.722;
   1:  PR[91,2] = PR[90,2] + 18.393;
   1:  PR[91,3] = PR[90,3] + 56.666;
   1:L PR[91] R[100]mm/sec CNT100;
   1:  PR[91,1] = PR[90,1] + -17.639;
   1:  PR[91,2] = PR[90,2] + 17.665;
   1:  PR[91,3] = PR[90,3] + 56.676;
   1:L PR[91] R[100]mm/sec CNT100;
   1:  PR[91,1] = PR[90,1] + -18.525;
   1:  PR[91,2] = PR[90,2] + 16.884;
   1:  PR[91,3] = PR[90,3] + 56.686;
   1:L PR[91] R[100]mm/sec CNT100;
   1:  PR[91,1] = PR[90,1] + -19.351;
   1:  PR[91,2] = PR[90,2] + 16.078;
   1:  PR[91,3] = PR[90,3] + 56.696;
   1:L PR[91] R[100]mm/sec CNT100;
   1:  PR[91,1] = PR[90,1] + -20.143;
   1:  PR[91,2] = PR[90,2] + 15.223;
   1:  PR[91,3] = PR[90,3] + 56.706;
   1:L PR[91] R[100]mm/sec CNT100;
   1:  PR[91,1] = PR[90,1] + -20.888;
   1:  PR[91,2] = PR[90,2] + 14.329;
   1:  PR[91,3] = PR[90,3] + 56.716;
   1:L PR[91] R[100]mm/sec CNT100;
   1:  PR[91,1] = PR[90,1] + -21.586;
   1:  PR[91,2] = PR[90,2] + 13.400;
   1:  PR[91,3] = PR[90,3] + 56.726;
   1:L PR[91] R[100]mm/sec CNT100;
   1:  PR[91,1] = PR[90,1] + -22.235;
   1:  PR[91,2] = PR[90,2] + 12.438;
   1:  PR[91,3] = PR[90,3] + 56.736;
   1:L PR[91] R[100]mm/sec CNT100;
   1:  PR[91,1] = PR[90,1] + -22.832;
   1:  PR[91,2] = PR[90,2] + 11.444;
   1:  PR[91,3] = PR[90,3] + 56.746;
   1:L PR[91] R[100]mm/sec CNT100;
   1:  PR[91,1] = PR[90,1] + -23.377;
   1:  PR[91,2] = PR[90,2] + 10.423;
   1:  PR[91,3] = PR[90,3] + 56.756;
   1:L PR[91] R[100]mm/sec CNT100;
   1:  PR[91,1] = PR[90,1] + -23.868;
   1:  PR[91,2] = PR[90,2] + 9.377;
   1:  PR[91,3] = PR[90,3] + 56.766;
   1:L PR[91] R[100]mm/sec CNT100;
   1:  PR[91,1] = PR[90,1] + -24.305;
   1:  PR[91,2] = PR[90,2] + 8.309;
   1:  PR[91,3] = PR[90,3] + 56.776;
   1:L PR[91] R[100]mm/sec CNT100;
   1:  PR[91,1] = PR[90,1] + -24.685;
   1:  PR[91,2] = PR[90,2] + 7.222;
   1:  PR[91,3] = PR[90,3] + 56.786;
   1:L PR[91] R[100]mm/sec CNT100;
   1:  PR[91,1] = PR[90,1] + -25.008;
   1:  PR[91,2] = PR[90,2] + 6.119;
   1:  PR[91,3] = PR[90,3] + 56.796;
   1:L PR[91] R[100]mm/sec CNT100;
   1:  PR[91,1] = PR[90,1] + -25.274;
   1:  PR[91,2] = PR[90,2] + 5.002;
   1:  PR[91,3] = PR[90,3] + 56.806;
   1:L PR[91] R[100]mm/sec CNT100;
   1:  PR[91,1] = PR[90,1] + -25.481;
   1:  PR[91,2] = PR[90,2] + 3.872;
   1:  PR[91,3] = PR[90,3] + 56.816;
   1:L PR[91] R[100]mm/sec CNT100;
   1:  PR[91,1] = PR[90,1] + -25.629;
   1:  PR[91,2] = PR[90,2] + 2.732;
   1:  PR[91,3] = PR[90,3] + 56.826;
   1:L PR[91] R[100]mm/sec CNT100;
   1:  PR[91,1] = PR[90,1] + -25.718;
   1:  PR[91,2] = PR[90,2] + 1.584;
   1:  PR[91,3] = PR[90,3] + 56.836;
   1:L PR[91] R[100]mm/sec CNT100;
   1:  PR[91,1] = PR[90,1] + -25.746;
   1:  PR[91,2] = PR[90,2] + 0.428;
   1:  PR[91,3] = PR[90,3] + 56.846;
   1:L PR[91] R[100]mm/sec CNT100;
   1:  PR[91,1] = PR[90,1] + -25.718;
   1:  PR[91,2] = PR[90,2] + -0.729;
   1:  PR[91,3] = PR[90,3] + 56.856;
   1:L PR[91] R[100]mm/sec CNT100;
   1:  PR[91,1] = PR[90,1] + -25.629;
   1:  PR[91,2] = PR[90,2] + -1.878;
   1:  PR[91,3] = PR[90,3] + 56.866;
   1:L PR[91] R[100]mm/sec CNT100;
   1:  PR[91,1] = PR[90,1] + -25.481;
   1:  PR[91,2] = PR[90,2] + -3.018;
   1:  PR[91,3] = PR[90,3] + 56.876;
   1:L PR[91] R[100]mm/sec CNT100;
   1:  PR[91,1] = PR[90,1] + -25.274;
   1:  PR[91,2] = PR[90,2] + -4.147;
   1:  PR[91,3] = PR[90,3] + 56.886;
   1:L PR[91] R[100]mm/sec CNT100;
   1:  PR[91,1] = PR[90,1] + -25.008;
   1:  PR[91,2] = PR[90,2] + -5.264;
   1:  PR[91,3] = PR[90,3] + 56.896;
   1:L PR[91] R[100]mm/sec CNT100;
   1:  PR[91,1] = PR[90,1] + -24.685;
   1:  PR[91,2] = PR[90,2] + -6.368;
   1:  PR[91,3] = PR[90,3] + 56.906;
   1:L PR[91] R[100]mm/sec CNT100;
   1:  PR[91,1] = PR[90,1] + -24.304;
   1:  PR[91,2] = PR[90,2] + -7.455;
   1:  PR[91,3] = PR[90,3] + 56.916;
   1:L PR[91] R[100]mm/sec CNT100;
   1:  PR[91,1] = PR[90,1] + -23.868;
   1:  PR[91,2] = PR[90,2] + -8.523;
   1:  PR[91,3] = PR[90,3] + 56.926;
   1:L PR[91] R[100]mm/sec CNT100;
   1:  PR[91,1] = PR[90,1] + -23.376;
   1:  PR[91,2] = PR[90,2] + -9.569;
   1:  PR[91,3] = PR[90,3] + 56.936;
   1:L PR[91] R[100]mm/sec CNT100;
   1:  PR[91,1] = PR[90,1] + -22.831;
   1:  PR[91,2] = PR[90,2] + -10.591;
   1:  PR[91,3] = PR[90,3] + 56.946;
   1:L PR[91] R[100]mm/sec CNT100;
   1:  PR[91,1] = PR[90,1] + -22.233;
   1:  PR[91,2] = PR[90,2] + -11.584;
   1:  PR[91,3] = PR[90,3] + 56.956;
   1:L PR[91] R[100]mm/sec CNT100;
   1:  PR[91,1] = PR[90,1] + -21.585;
   1:  PR[91,2] = PR[90,2] + -12.547;
   1:  PR[91,3] = PR[90,3] + 56.966;
   1:L PR[91] R[100]mm/sec CNT100;
   1:  PR[91,1] = PR[90,1] + -20.887;
   1:  PR[91,2] = PR[90,2] + -13.476;
   1:  PR[91,3] = PR[90,3] + 56.976;
   1:L PR[91] R[100]mm/sec CNT100;
   1:  PR[91,1] = PR[90,1] + -20.141;
   1:  PR[91,2] = PR[90,2] + -14.370;
   1:  PR[91,3] = PR[90,3] + 56.986;
   1:L PR[91] R[100]mm/sec CNT100;
   1:  PR[91,1] = PR[90,1] + -19.344;
   1:  PR[91,2] = PR[90,2] + -15.230;
   1:  PR[91,3] = PR[90,3] + 56.996;
   1:L PR[91] R[100]mm/sec CNT100;
   1:  PR[91,1] = PR[90,1] + -18.514;
   1:  PR[91,2] = PR[90,2] + -16.039;
   1:  PR[91,3] = PR[90,3] + 57.006;
   1:L PR[91] R[100]mm/sec CNT100;
   1:  PR[91,1] = PR[90,1] + -17.637;
   1:  PR[91,2] = PR[90,2] + -16.812;
   1:  PR[91,3] = PR[90,3] + 57.016;
   1:L PR[91] R[100]mm/sec CNT100;
   1:  PR[91,1] = PR[90,1] + -16.720;
   1:  PR[91,2] = PR[90,2] + -17.540;
   1:  PR[91,3] = PR[90,3] + 57.026;
   1:L PR[91] R[100]mm/sec CNT100;
   1:  PR[91,1] = PR[90,1] + -15.766;
   1:  PR[91,2] = PR[90,2] + -18.222;
   1:  PR[91,3] = PR[90,3] + 57.036;
   1:L PR[91] R[100]mm/sec CNT100;
   1:  PR[91,1] = PR[90,1] + -14.776;
   1:  PR[91,2] = PR[90,2] + -18.855;
   1:  PR[91,3] = PR[90,3] + 57.046;
   1:L PR[91] R[100]mm/sec CNT100;
   1:  PR[91,1] = PR[90,1] + -13.755;
   1:  PR[91,2] = PR[90,2] + -19.437;
   1:  PR[91,3] = PR[90,3] + 57.057;
   1:L PR[91] R[100]mm/sec CNT100;
   1:  PR[91,1] = PR[90,1] + -12.704;
   1:  PR[91,2] = PR[90,2] + -19.968;
   1:  PR[91,3] = PR[90,3] + 57.067;
   1:L PR[91] R[100]mm/sec CNT100;
   1:  PR[91,1] = PR[90,1] + -11.626;
   1:  PR[91,2] = PR[90,2] + -20.444;
   1:  PR[91,3] = PR[90,3] + 57.077;
   1:L PR[91] R[100]mm/sec CNT100;
   1:  PR[91,1] = PR[90,1] + -10.524;
   1:  PR[91,2] = PR[90,2] + -20.866;
   1:  PR[91,3] = PR[90,3] + 57.087;
   1:L PR[91] R[100]mm/sec CNT100;
   1:  PR[91,1] = PR[90,1] + -9.400;
   1:  PR[91,2] = PR[90,2] + -21.232;
   1:  PR[91,3] = PR[90,3] + 57.097;
   1:L PR[91] R[100]mm/sec CNT100;
   1:  PR[91,1] = PR[90,1] + -8.258;
   1:  PR[91,2] = PR[90,2] + -21.540;
   1:  PR[91,3] = PR[90,3] + 57.108;
   1:L PR[91] R[100]mm/sec CNT100;
   1:  PR[91,1] = PR[90,1] + -7.357;
   1:  PR[91,2] = PR[90,2] + -21.736;
   1:  PR[91,3] = PR[90,3] + 57.118;
   1:L PR[91] R[100]mm/sec CNT100;
   1:  PR[91,1] = PR[90,1] + -7.103;
   1:  PR[91,2] = PR[90,2] + -21.789;
   1:  PR[91,3] = PR[90,3] + 57.126;
   1:L PR[91] R[100]mm/sec CNT100;
   1:  PR[91,1] = PR[90,1] + -5.932;
   1:  PR[91,2] = PR[90,2] + -21.980;
   1:  PR[91,3] = PR[90,3] + 57.128;
   1:L PR[91] R[100]mm/sec CNT100;
   1:  PR[91,1] = PR[90,1] + -4.754;
   1:  PR[91,2] = PR[90,2] + -22.111;
   1:  PR[91,3] = PR[90,3] + 57.138;
   1:L PR[91] R[100]mm/sec CNT100;
   1:  PR[91,1] = PR[90,1] + -3.569;
   1:  PR[91,2] = PR[90,2] + -22.181;
   1:  PR[91,3] = PR[90,3] + 57.148;
   1:L PR[91] R[100]mm/sec CNT100;
   1:  PR[91,1] = PR[90,1] + -2.383;
   1:  PR[91,2] = PR[90,2] + -22.190;
   1:  PR[91,3] = PR[90,3] + 57.159;
   1:L PR[91] R[100]mm/sec CNT100;
   1:  PR[91,1] = PR[90,1] + -1.195;
   1:  PR[91,2] = PR[90,2] + -22.139;
   1:  PR[91,3] = PR[90,3] + 57.169;
   1:L PR[91] R[100]mm/sec CNT100;
   1:  PR[91,1] = PR[90,1] + -0.400;
   1:  PR[91,2] = PR[90,2] + -22.067;
